LIN {X 0,Y 426.116,Z 779.168,A -85,B 0,C 180,E1 -10324.509,E2 -10324.509} C_VEL
LIN {X 0,Y 425.527,Z 793.819,A -85,B 0,C 180,E1 -10324.947,E2 -10324.947} C_VEL
LIN {X 0,Y 424.719,Z 807.739,A -85,B 0,C 180,E1 -10325.563,E2 -10325.563} C_VEL
LIN {X 0,Y 423.969,Z 820.23,A -85,B 0,C 180,E1 -10326.308,E2 -10326.308} C_VEL
LIN {X 0,Y 422.947,Z 832.999,A -85,B 0,C 180,E1 -10327.273,E2 -10327.273} C_VEL
LIN {X 0,Y 422.02,Z 844.698,A -85,B 0,C 180,E1 -10328.38,E2 -10328.38} C_VEL
LIN {X 0,Y 421.156,Z 854.395,A -85,B 0,C 180,E1 -10329.486,E2 -10329.486} C_VEL
LIN {X 0,Y 420.11,Z 865.116,A -85,B 0,C 180,E1 -10330.961,E2 -10330.961} C_VEL
LIN {X 0,Y 419.261,Z 873.928,A -85,B 0,C 180,E1 -10332.438,E2 -10332.438} C_VEL
LIN {X 0,Y 418.634,Z 881.226,A -85,B 0,C 180,E1 -10333.919,E2 -10333.919} C_VEL
LIN {X 0,Y 417.959,Z 888.478,A -85,B 0,C 180,E1 -10335.723,E2 -10335.723} C_VEL
LIN {X 0,Y 417.146,Z 891.035,A -85,B 0,C 180,E1 -10336.445,E2 -10336.445} C_VEL
LIN {X 0,Y 414.039,Z 894.793,A -85,B 0,C 180,E1 -10337.635,E2 -10337.635} C_VEL
LIN {X 0,Y 411.432,Z 897.379,A -85,B 0,C 180,E1 -10338.619,E2 -10338.619} C_VEL
LIN {X 0,Y 410.263,Z 899.081,A -85,B 0,C 180,E1 -10339.397,E2 -10339.397} C_VEL
LIN {X 0,Y 410.139,Z 899.54,A -85,B 0,C 180,E1 -10339.664,E2 -10339.664} C_VEL
LIN {X 0,Y 410.039,Z 901.862,A -85,B 0,C 180,E1 -10341.126,E2 -10341.126} C_VEL
LIN {X 0,Y 410.034,Z 903.737,A -85,B 0,C 180,E1 -10343.109,E2 -10343.109} C_VEL
LIN {X 0,Y 409.968,Z 904.281,A -85,B 0,C 180,E1 -10345.083,E2 -10345.083} C_VEL
LIN {X 0,Y 409.988,Z 903.511,A -85,B 0,C 180,E1 -10347.052,E2 -10347.052} C_VEL
LIN {X 0,Y 410.005,Z 901.424,A -85,B 0,C 180,E1 -10349.018,E2 -10349.018} C_VEL
LIN {X 0,Y 410.11,Z 897.97,A -85,B 0,C 180,E1 -10350.982,E2 -10350.982} C_VEL
LIN {X 0,Y 410.446,Z 893.043,A -85,B 0,C 180,E1 -10352.945,E2 -10352.945} C_VEL
LIN {X 0,Y 411.09,Z 886.486,A -85,B 0,C 180,E1 -10354.904,E2 -10354.904} C_VEL
LIN {X 0,Y 411.743,Z 879.197,A -85,B 0,C 180,E1 -10356.616,E2 -10356.616} C_VEL
LIN {X 0,Y 412.336,Z 870.804,A -85,B 0,C 180,E1 -10358.222,E2 -10358.222} C_VEL
LIN {X 0,Y 413.209,Z 861.976,A -85,B 0,C 180,E1 -10359.614,E2 -10359.614} C_VEL
LIN {X 0,Y 414.215,Z 851.288,A -85,B 0,C 180,E1 -10361.004,E2 -10361.004} C_VEL
LIN {X 0,Y 415.185,Z 839.942,A -85,B 0,C 180,E1 -10362.216,E2 -10362.216} C_VEL
LIN {X 0,Y 416.148,Z 827.376,A -85,B 0,C 180,E1 -10363.303,E2 -10363.303} C_VEL
LIN {X 0,Y 416.988,Z 815.158,A -85,B 0,C 180,E1 -10364.146,E2 -10364.146} C_VEL
LIN {X 0,Y 417.734,Z 801.639,A -85,B 0,C 180,E1 -10364.867,E2 -10364.867} C_VEL
LIN {X 0,Y 418.279,Z 787.615,A -85,B 0,C 180,E1 -10365.408,E2 -10365.408} C_VEL
LIN {X 0,Y 418.632,Z 772.8,A -85,B 0,C 180,E1 -10365.769,E2 -10365.769} C_VEL
LIN {X 0,Y 420.223,Z 667.238,A -85,B 0,C 180,E1 -10367.579,E2 -10367.579} C_VEL
LIN {X 0,Y 416.862,Z 653.116,A -85,B 0,C 180,E1 -10368.014,E2 -10368.014} C_VEL
LIN {X 0,Y 413.362,Z 643.418,A -85,B 0,C 180,E1 -10368.406,E2 -10368.406} C_VEL
LIN {X 0,Y 411.214,Z 633.392,A -85,B 0,C 180,E1 -10370.775,E2 -10370.775} C_VEL
LIN {X 0,Y 411.193,Z 633.392,A -85,B 0,C 180,E1 -10374.218,E2 -10374.218} C_VEL
LIN {X 0,Y 411.145,Z 633.397,A -85,B 0,C 180,E1 -10377.486,E2 -10377.486} C_VEL
LIN {X 0,Y 411.197,Z 633.388,A -85,B 0,C 180,E1 -10379.713,E2 -10379.713} C_VEL
LIN {X 0,Y 411.206,Z 633.39,A -85,B 0,C 180,E1 -10383.156,E2 -10383.156} C_VEL
LIN {X 0,Y 411.192,Z 633.39,A -85,B 0,C 180,E1 -10386.551,E2 -10386.551} C_VEL
LIN {X 0,Y 411.171,Z 633.379,A -85,B 0,C 180,E1 -10389.72,E2 -10389.72} C_VEL
LIN {X 0,Y 411.165,Z 633.393,A -85,B 0,C 180,E1 -10393.135,E2 -10393.135} C_VEL
LIN {X 0,Y 411.167,Z 633.39,A -85,B 0,C 180,E1 -10395.882,E2 -10395.882} C_VEL
LIN {X 0,Y 411.161,Z 633.392,A -85,B 0,C 180,E1 -10399.493,E2 -10399.493} C_VEL
LIN {X 0,Y 411.186,Z 633.373,A -85,B 0,C 180,E1 -10402.025,E2 -10402.025} C_VEL
LIN {X 0,Y 411.207,Z 633.387,A -85,B 0,C 180,E1 -10405.666,E2 -10405.666} C_VEL
LIN {X 0,Y 411.192,Z 633.385,A -85,B 0,C 180,E1 -10409.152,E2 -10409.152} C_VEL
LIN {X 0,Y 411.183,Z 633.39,A -85,B 0,C 180,E1 -10411.407,E2 -10411.407} C_VEL
LIN {X 0,Y 411.215,Z 633.383,A -85,B 0,C 180,E1 -10414.934,E2 -10414.934} C_VEL
LIN {X 0,Y 411.206,Z 633.386,A -85,B 0,C 180,E1 -10417.913,E2 -10417.913} C_VEL
LIN {X 0,Y 411.223,Z 633.383,A -85,B 0,C 180,E1 -10421.051,E2 -10421.051} C_VEL
LIN {X 0,Y 411.257,Z 633.377,A -85,B 0,C 180,E1 -10424.131,E2 -10424.131} C_VEL
LIN {X 0,Y 411.307,Z 633.374,A -85,B 0,C 180,E1 -10427.165,E2 -10427.165} C_VEL
LIN {X 0,Y 411.294,Z 633.368,A -85,B 0,C 180,E1 -10430.161,E2 -10430.161} C_VEL
LIN {X 0,Y 411.396,Z 633.362,A -85,B 0,C 180,E1 -10433.132,E2 -10433.132} C_VEL
LIN {X 0,Y 411.305,Z 633.372,A -85,B 0,C 180,E1 -10435.099,E2 -10435.099} C_VEL
LIN {X 0,Y 411.512,Z 633.351,A -85,B 0,C 180,E1 -10438.042,E2 -10438.042} C_VEL
LIN {X 0,Y 411.641,Z 633.33,A -85,B 0,C 180,E1 -10440,E2 -10440} C_VEL
LIN {X 0,Y 411.459,Z 633.353,A -85,B 0,C 180,E1 -10442.937,E2 -10442.937} C_VEL
LIN {X 0,Y 411.432,Z 633.354,A -85,B 0,C 180,E1 -10446.867,E2 -10446.867} C_VEL
LIN {X 0,Y 411.295,Z 633.377,A -85,B 0,C 180,E1 -10449.838,E2 -10449.838} C_VEL
LIN {X 0,Y 411.308,Z 633.372,A -85,B 0,C 180,E1 -10453.104,E2 -10453.104} C_VEL
LIN {X 0,Y 411.267,Z 633.376,A -85,B 0,C 180,E1 -10456.869,E2 -10456.869} C_VEL
LIN {X 0,Y 411.233,Z 633.381,A -85,B 0,C 180,E1 -10459.986,E2 -10459.986} C_VEL
LIN {X 0,Y 411.198,Z 633.382,A -85,B 0,C 180,E1 -10463.148,E2 -10463.148} C_VEL
LIN {X 0,Y 411.238,Z 633.382,A -85,B 0,C 180,E1 -10466.381,E2 -10466.381} C_VEL
LIN {X 0,Y 411.202,Z 633.386,A -85,B 0,C 180,E1 -10469.712,E2 -10469.712} C_VEL
LIN {X 0,Y 411.208,Z 633.384,A -85,B 0,C 180,E1 -10473.155,E2 -10473.155} C_VEL
LIN {X 0,Y 411.197,Z 633.389,A -85,B 0,C 180,E1 -10476.553,E2 -10476.553} C_VEL
LIN {X 0,Y 411.228,Z 633.381,A -85,B 0,C 180,E1 -10479.73,E2 -10479.73} C_VEL
LIN {X 0,Y 411.178,Z 633.389,A -85,B 0,C 180,E1 -10483.133,E2 -10483.133} C_VEL
LIN {X 0,Y 411.174,Z 633.389,A -85,B 0,C 180,E1 -10485.88,E2 -10485.88} C_VEL
LIN {X 0,Y 411.167,Z 633.394,A -85,B 0,C 180,E1 -10488.771,E2 -10488.771} C_VEL
LIN {X 0,Y 411.213,Z 633.386,A -85,B 0,C 180,E1 -10491.83,E2 -10491.83} C_VEL
LIN {X 0,Y 411.213,Z 633.39,A -85,B 0,C 180,E1 -10495.121,E2 -10495.121} C_VEL
LIN {X 0,Y 411.167,Z 633.39,A -85,B 0,C 180,E1 -10498.003,E2 -10498.003} C_VEL
LIN {X 0,Y 411.262,Z 633.533,A -85,B 0,C 180,E1 -10499.372,E2 -10499.372} C_VEL
LIN {X 0,Y 414.549,Z 647.989,A -85,B 0,C 180,E1 -10502.318,E2 -10502.318} C_VEL
LIN {X 0,Y 415.856,Z 654.509,A -85,B 0,C 180,E1 -10503.599,E2 -10503.599} C_VEL
LIN {X 0,Y 414.842,Z 669.698,A -85,B 0,C 180,E1 -10506.317,E2 -10506.317} C_VEL
LIN {X 0,Y 414.706,Z 671.836,A -85,B 0,C 180,E1 -10506.696,E2 -10506.696} C_VEL
LIN {X 0,Y 419.881,Z 702.214,A -85,B 0,C 180,E1 -10507.528,E2 -10507.528} C_VEL
LIN {X 0,Y 418.525,Z 800.905,A -85,B 0,C 180,E1 -10509.223,E2 -10509.223} C_VEL
LIN {X 0,Y 418.065,Z 815.953,A -85,B 0,C 180,E1 -10509.552,E2 -10509.552} C_VEL
LIN {X 0,Y 417.398,Z 830.189,A -85,B 0,C 180,E1 -10510.064,E2 -10510.064} C_VEL
LIN {X 0,Y 416.641,Z 843.346,A -85,B 0,C 180,E1 -10510.731,E2 -10510.731} C_VEL
LIN {X 0,Y 415.764,Z 855.462,A -85,B 0,C 180,E1 -10511.521,E2 -10511.521} C_VEL
LIN {X 0,Y 414.818,Z 867.42,A -85,B 0,C 180,E1 -10512.499,E2 -10512.499} C_VEL
LIN {X 0,Y 413.753,Z 879.543,A -85,B 0,C 180,E1 -10513.724,E2 -10513.724} C_VEL
LIN {X 0,Y 412.833,Z 889.574,A -85,B 0,C 180,E1 -10514.953,E2 -10514.953} C_VEL
LIN {X 0,Y 411.997,Z 899.202,A -85,B 0,C 180,E1 -10516.373,E2 -10516.373} C_VEL
LIN {X 0,Y 411.326,Z 907.866,A -85,B 0,C 180,E1 -10517.918,E2 -10517.918} C_VEL
LIN {X 0,Y 410.685,Z 915.798,A -85,B 0,C 180,E1 -10519.648,E2 -10519.648} C_VEL
LIN {X 0,Y 410.353,Z 921.358,A -85,B 0,C 180,E1 -10521.133,E2 -10521.133} C_VEL
LIN {X 0,Y 410.085,Z 927.19,A -85,B 0,C 180,E1 -10523.11,E2 -10523.11} C_VEL
LIN {X 0,Y 409.995,Z 931.435,A -85,B 0,C 180,E1 -10525.083,E2 -10525.083} C_VEL
LIN {X 0,Y 409.934,Z 934.224,A -85,B 0,C 180,E1 -10527.052,E2 -10527.052} C_VEL
LIN {X 0,Y 409.991,Z 935.101,A -85,B 0,C 180,E1 -10528.035,E2 -10528.035} C_VEL
LIN {X 0,Y 409.946,Z 935.837,A -85,B 0,C 180,E1 -10530,E2 -10530} C_VEL
LIN {X 0,Y 409.99,Z 935.235,A -85,B 0,C 180,E1 -10531.965,E2 -10531.965} C_VEL
LIN {X 0,Y 409.924,Z 933.276,A -85,B 0,C 180,E1 -10533.932,E2 -10533.932} C_VEL
LIN {X 0,Y 410.042,Z 929.917,A -85,B 0,C 180,E1 -10535.903,E2 -10535.903} C_VEL
LIN {X 0,Y 410.188,Z 925.062,A -85,B 0,C 180,E1 -10537.878,E2 -10537.878} C_VEL
LIN {X 0,Y 410.612,Z 918.581,A -85,B 0,C 180,E1 -10539.855,E2 -10539.855} C_VEL
LIN {X 0,Y 411.17,Z 911.384,A -85,B 0,C 180,E1 -10541.586,E2 -10541.586} C_VEL
LIN {X 0,Y 411.87,Z 903.781,A -85,B 0,C 180,E1 -10543.083,E2 -10543.083} C_VEL
LIN {X 0,Y 412.602,Z 894.853,A -85,B 0,C 180,E1 -10544.551,E2 -10544.551} C_VEL
LIN {X 0,Y 413.688,Z 883.963,A -85,B 0,C 180,E1 -10546.025,E2 -10546.025} C_VEL
LIN {X 0,Y 414.754,Z 872.932,A -85,B 0,C 180,E1 -10547.25,E2 -10547.25} C_VEL
LIN {X 0,Y 415.898,Z 860.846,A -85,B 0,C 180,E1 -10548.345,E2 -10548.345} C_VEL
LIN {X 0,Y 416.982,Z 847.686,A -85,B 0,C 180,E1 -10549.292,E2 -10549.292} C_VEL
LIN {X 0,Y 417.882,Z 834.246,A -85,B 0,C 180,E1 -10550.04,E2 -10550.04} C_VEL
LIN {X 0,Y 418.672,Z 820.158,A -85,B 0,C 180,E1 -10550.609,E2 -10550.609} C_VEL
LIN {X 0,Y 419.235,Z 805.296,A -85,B 0,C 180,E1 -10550.997,E2 -10550.997} C_VEL
LIN {X 0,Y 420.84,Z 702.534,A -85,B 0,C 180,E1 -10552.785,E2 -10552.785} C_VEL
LIN {X 0,Y 416.253,Z 677.29,A -85,B 0,C 180,E1 -10553.539,E2 -10553.539} C_VEL
LIN {X 0,Y 415.169,Z 671.541,A -85,B 0,C 180,E1 -10553.744,E2 -10553.744} C_VEL
LIN {X 0,Y 416.408,Z 657.156,A -85,B 0,C 180,E1 -10556.357,E2 -10556.357} C_VEL
LIN {X 0,Y 415.295,Z 650.459,A -85,B 0,C 180,E1 -10557.704,E2 -10557.704} C_VEL
LIN {X 0,Y 412.202,Z 637.376,A -85,B 0,C 180,E1 -10560.484,E2 -10560.484} C_VEL
LIN {X 0,Y 411.169,Z 633.391,A -85,B 0,C 180,E1 -10561.395,E2 -10561.395} C_VEL
LIN {X 0,Y 411.207,Z 633.383,A -85,B 0,C 180,E1 -10564.333,E2 -10564.333} C_VEL
LIN {X 0,Y 411.203,Z 633.386,A -85,B 0,C 180,E1 -10567.973,E2 -10567.973} C_VEL
LIN {X 0,Y 411.201,Z 633.385,A -85,B 0,C 180,E1 -10571.234,E2 -10571.234} C_VEL
LIN {X 0,Y 411.18,Z 633.385,A -85,B 0,C 180,E1 -10574.49,E2 -10574.49} C_VEL
LIN {X 0,Y 411.199,Z 633.38,A -85,B 0,C 180,E1 -10578.197,E2 -10578.197} C_VEL
LIN {X 0,Y 411.232,Z 633.383,A -85,B 0,C 180,E1 -10580.778,E2 -10580.778} C_VEL
LIN {X 0,Y 411.201,Z 633.385,A -85,B 0,C 180,E1 -10584.472,E2 -10584.472} C_VEL
LIN {X 0,Y 411.207,Z 633.382,A -85,B 0,C 180,E1 -10586.873,E2 -10586.873} C_VEL
LIN {X 0,Y 411.233,Z 633.379,A -85,B 0,C 180,E1 -10590.644,E2 -10590.644} C_VEL
LIN {X 0,Y 411.239,Z 633.381,A -85,B 0,C 180,E1 -10593.619,E2 -10593.619} C_VEL
LIN {X 0,Y 411.204,Z 633.382,A -85,B 0,C 180,E1 -10596.853,E2 -10596.853} C_VEL
LIN {X 0,Y 411.217,Z 633.388,A -85,B 0,C 180,E1 -10600.05,E2 -10600.05} C_VEL
LIN {X 0,Y 411.266,Z 633.377,A -85,B 0,C 180,E1 -10603.131,E2 -10603.131} C_VEL
LIN {X 0,Y 411.307,Z 633.37,A -85,B 0,C 180,E1 -10606.896,E2 -10606.896} C_VEL
LIN {X 0,Y 411.295,Z 633.373,A -85,B 0,C 180,E1 -10610.162,E2 -10610.162} C_VEL
LIN {X 0,Y 411.454,Z 633.354,A -85,B 0,C 180,E1 -10613.133,E2 -10613.133} C_VEL
LIN {X 0,Y 411.311,Z 633.367,A -85,B 0,C 180,E1 -10615.099,E2 -10615.099} C_VEL
LIN {X 0,Y 411.513,Z 633.35,A -85,B 0,C 180,E1 -10618.043,E2 -10618.043} C_VEL
LIN {X 0,Y 411.642,Z 633.332,A -85,B 0,C 180,E1 -10620,E2 -10620} C_VEL
LIN {X 0,Y 411.459,Z 633.355,A -85,B 0,C 180,E1 -10622.938,E2 -10622.938} C_VEL
LIN {X 0,Y 411.453,Z 633.357,A -85,B 0,C 180,E1 -10626.867,E2 -10626.867} C_VEL
LIN {X 0,Y 411.294,Z 633.372,A -85,B 0,C 180,E1 -10629.839,E2 -10629.839} C_VEL
LIN {X 0,Y 411.308,Z 633.373,A -85,B 0,C 180,E1 -10633.105,E2 -10633.105} C_VEL
LIN {X 0,Y 411.265,Z 633.383,A -85,B 0,C 180,E1 -10636.869,E2 -10636.869} C_VEL
LIN {X 0,Y 411.233,Z 633.377,A -85,B 0,C 180,E1 -10639.987,E2 -10639.987} C_VEL
LIN {X 0,Y 411.198,Z 633.384,A -85,B 0,C 180,E1 -10643.148,E2 -10643.148} C_VEL
LIN {X 0,Y 411.198,Z 633.389,A -85,B 0,C 180,E1 -10646.384,E2 -10646.384} C_VEL
LIN {X 0,Y 411.2,Z 633.374,A -85,B 0,C 180,E1 -10649.713,E2 -10649.713} C_VEL
LIN {X 0,Y 411.209,Z 633.386,A -85,B 0,C 180,E1 -10653.156,E2 -10653.156} C_VEL
LIN {X 0,Y 411.194,Z 633.389,A -85,B 0,C 180,E1 -10656.553,E2 -10656.553} C_VEL
LIN {X 0,Y 411.18,Z 633.384,A -85,B 0,C 180,E1 -10659.722,E2 -10659.722} C_VEL
LIN {X 0,Y 411.167,Z 633.397,A -85,B 0,C 180,E1 -10663.135,E2 -10663.135} C_VEL
LIN {X 0,Y 411.166,Z 633.389,A -85,B 0,C 180,E1 -10665.882,E2 -10665.882} C_VEL
LIN {X 0,Y 411.165,Z 633.397,A -85,B 0,C 180,E1 -10669.494,E2 -10669.494} C_VEL
LIN {X 0,Y 411.19,Z 633.391,A -85,B 0,C 180,E1 -10672.026,E2 -10672.026} C_VEL
LIN {X 0,Y 411.196,Z 633.39,A -85,B 0,C 180,E1 -10675.666,E2 -10675.666} C_VEL
LIN {X 0,Y 411.209,Z 633.511,A -85,B 0,C 180,E1 -10678.711,E2 -10678.711} C_VEL
LIN {X 0,Y 413.516,Z 643.651,A -85,B 0,C 180,E1 -10681.219,E2 -10681.219} C_VEL
LIN {X 0,Y 418.909,Z 657.328,A -85,B 0,C 180,E1 -10681.84,E2 -10681.84} C_VEL
LIN {X 0,Y 421.274,Z 668.298,A -85,B 0,C 180,E1 -10682.193,E2 -10682.193} C_VEL
LIN {X 0,Y 419.565,Z 779.554,A -85,B 0,C 180,E1 -10684.149,E2 -10684.149} C_VEL
LIN {X 0,Y 418.987,Z 793.733,A -85,B 0,C 180,E1 -10684.577,E2 -10684.577} C_VEL
LIN {X 0,Y 418.213,Z 806.917,A -85,B 0,C 180,E1 -10685.158,E2 -10685.158} C_VEL
LIN {X 0,Y 417.367,Z 819.977,A -85,B 0,C 180,E1 -10685.935,E2 -10685.935} C_VEL
LIN {X 0,Y 416.313,Z 832.576,A -85,B 0,C 180,E1 -10686.89,E2 -10686.89} C_VEL
LIN {X 0,Y 415.287,Z 844.394,A -85,B 0,C 180,E1 -10688.011,E2 -10688.011} C_VEL
LIN {X 0,Y 414.397,Z 854.189,A -85,B 0,C 180,E1 -10689.136,E2 -10689.136} C_VEL
LIN {X 0,Y 413.297,Z 864.988,A -85,B 0,C 180,E1 -10690.635,E2 -10690.635} C_VEL
LIN {X 0,Y 412.366,Z 873.867,A -85,B 0,C 180,E1 -10692.135,E2 -10692.135} C_VEL
LIN {X 0,Y 411.691,Z 881.223,A -85,B 0,C 180,E1 -10693.64,E2 -10693.64} C_VEL
LIN {X 0,Y 411.075,Z 887.322,A -85,B 0,C 180,E1 -10695.141,E2 -10695.141} C_VEL
LIN {X 0,Y 410.691,Z 892.354,A -85,B 0,C 180,E1 -10696.643,E2 -10696.643} C_VEL
LIN {X 0,Y 410.304,Z 897.512,A -85,B 0,C 180,E1 -10698.64,E2 -10698.64} C_VEL
LIN {X 0,Y 410.139,Z 899.54,A -85,B 0,C 180,E1 -10699.664,E2 -10699.664} C_VEL
LIN {X 0,Y 409.406,Z 900.948,A -85,B 0,C 180,E1 -10700.459,E2 -10700.459} C_VEL
LIN {X 0,Y 406.562,Z 902.765,A -85,B 0,C 180,E1 -10701.765,E2 -10701.765} C_VEL
LIN {X 0,Y 404.149,Z 903.807,A -85,B 0,C 180,E1 -10702.829,E2 -10702.829} C_VEL
LIN {X 0,Y 403.043,Z 904.3,A -85,B 0,C 180,E1 -10703.655,E2 -10703.655} C_VEL
LIN {X 0,Y 402.912,Z 904.415,A -85,B 0,C 180,E1 -10703.935,E2 -10703.935} C_VEL
LIN {X 0,Y 402.838,Z 904.364,A -85,B 0,C 180,E1 -10705.998,E2 -10705.998} C_VEL
LIN {X 0,Y 402.959,Z 902.973,A -85,B 0,C 180,E1 -10708.001,E2 -10708.001} C_VEL
LIN {X 0,Y 402.947,Z 900.255,A -85,B 0,C 180,E1 -10710,E2 -10710} C_VEL
LIN {X 0,Y 403.191,Z 897.316,A -85,B 0,C 180,E1 -10711.498,E2 -10711.498} C_VEL
LIN {X 0,Y 403.618,Z 892.036,A -85,B 0,C 180,E1 -10713.494,E2 -10713.494} C_VEL
LIN {X 0,Y 404.05,Z 886.977,A -85,B 0,C 180,E1 -10714.989,E2 -10714.989} C_VEL
LIN {X 0,Y 404.729,Z 879.746,A -85,B 0,C 180,E1 -10716.731,E2 -10716.731} C_VEL
LIN {X 0,Y 405.318,Z 871.709,A -85,B 0,C 180,E1 -10718.314,E2 -10718.314} C_VEL
LIN {X 0,Y 406.177,Z 863.265,A -85,B 0,C 180,E1 -10719.687,E2 -10719.687} C_VEL
LIN {X 0,Y 407.117,Z 854.045,A -85,B 0,C 180,E1 -10720.947,E2 -10720.947} C_VEL
LIN {X 0,Y 408.115,Z 843.248,A -85,B 0,C 180,E1 -10722.178,E2 -10722.178} C_VEL
LIN {X 0,Y 409.041,Z 831.435,A -85,B 0,C 180,E1 -10723.286,E2 -10723.286} C_VEL
LIN {X 0,Y 410.04,Z 818.329,A -85,B 0,C 180,E1 -10724.264,E2 -10724.264} C_VEL
LIN {X 0,Y 410.89,Z 804.421,A -85,B 0,C 180,E1 -10725.057,E2 -10725.057} C_VEL
LIN {X 0,Y 411.522,Z 790.504,A -85,B 0,C 180,E1 -10725.635,E2 -10725.635} C_VEL
LIN {X 0,Y 411.884,Z 775.94,A -85,B 0,C 180,E1 -10726.034,E2 -10726.034} C_VEL
LIN {X 0,Y 413.626,Z 668.286,A -85,B 0,C 180,E1 -10727.915,E2 -10727.915} C_VEL
LIN {X 0,Y 410.4,Z 655.06,A -85,B 0,C 180,E1 -10728.336,E2 -10728.336} C_VEL
LIN {X 0,Y 406.21,Z 643.728,A -85,B 0,C 180,E1 -10728.802,E2 -10728.802} C_VEL
LIN {X 0,Y 404.161,Z 634.27,A -85,B 0,C 180,E1 -10731.084,E2 -10731.084} C_VEL
LIN {X 0,Y 404.152,Z 634.268,A -85,B 0,C 180,E1 -10733.576,E2 -10733.576} C_VEL
LIN {X 0,Y 404.1,Z 634.275,A -85,B 0,C 180,E1 -10736.884,E2 -10736.884} C_VEL
LIN {X 0,Y 404.144,Z 634.269,A -85,B 0,C 180,E1 -10740.285,E2 -10740.285} C_VEL
LIN {X 0,Y 404.139,Z 634.267,A -85,B 0,C 180,E1 -10743.813,E2 -10743.813} C_VEL
LIN {X 0,Y 404.135,Z 634.271,A -85,B 0,C 180,E1 -10746.874,E2 -10746.874} C_VEL
LIN {X 0,Y 404.12,Z 634.256,A -85,B 0,C 180,E1 -10750.075,E2 -10750.075} C_VEL
LIN {X 0,Y 404.145,Z 634.268,A -85,B 0,C 180,E1 -10753.082,E2 -10753.082} C_VEL
LIN {X 0,Y 404.123,Z 634.267,A -85,B 0,C 180,E1 -10755.922,E2 -10755.922} C_VEL
LIN {X 0,Y 404.104,Z 634.271,A -85,B 0,C 180,E1 -10758.632,E2 -10758.632} C_VEL
LIN {X 0,Y 404.141,Z 634.254,A -85,B 0,C 180,E1 -10761.495,E2 -10761.495} C_VEL
LIN {X 0,Y 404.182,Z 634.255,A -85,B 0,C 180,E1 -10764.983,E2 -10764.983} C_VEL
LIN {X 0,Y 404.142,Z 634.263,A -85,B 0,C 180,E1 -10768.442,E2 -10768.442} C_VEL
LIN {X 0,Y 404.156,Z 634.259,A -85,B 0,C 180,E1 -10770.862,E2 -10770.862} C_VEL
LIN {X 0,Y 404.141,Z 634.262,A -85,B 0,C 180,E1 -10774.23,E2 -10774.23} C_VEL
LIN {X 0,Y 404.169,Z 634.262,A -85,B 0,C 180,E1 -10777.508,E2 -10777.508} C_VEL
LIN {X 0,Y 404.166,Z 634.26,A -85,B 0,C 180,E1 -10780.707,E2 -10780.707} C_VEL
LIN {X 0,Y 404.224,Z 634.255,A -85,B 0,C 180,E1 -10783.848,E2 -10783.848} C_VEL
LIN {X 0,Y 404.286,Z 634.247,A -85,B 0,C 180,E1 -10786.939,E2 -10786.939} C_VEL
LIN {X 0,Y 404.259,Z 634.244,A -85,B 0,C 180,E1 -10789.988,E2 -10789.988} C_VEL
LIN {X 0,Y 404.346,Z 634.24,A -85,B 0,C 180,E1 -10793.011,E2 -10793.011} C_VEL
LIN {X 0,Y 404.275,Z 634.247,A -85,B 0,C 180,E1 -10795.013,E2 -10795.013} C_VEL
LIN {X 0,Y 404.481,Z 634.227,A -85,B 0,C 180,E1 -10798.008,E2 -10798.008} C_VEL
LIN {X 0,Y 404.61,Z 634.206,A -85,B 0,C 180,E1 -10800,E2 -10800} C_VEL
LIN {X 0,Y 404.417,Z 634.23,A -85,B 0,C 180,E1 -10802.988,E2 -10802.988} C_VEL
LIN {X 0,Y 404.382,Z 634.233,A -85,B 0,C 180,E1 -10806.987,E2 -10806.987} C_VEL
LIN {X 0,Y 404.26,Z 634.251,A -85,B 0,C 180,E1 -10810.011,E2 -10810.011} C_VEL
LIN {X 0,Y 404.269,Z 634.249,A -85,B 0,C 180,E1 -10813.211,E2 -10813.211} C_VEL
LIN {X 0,Y 404.221,Z 634.253,A -85,B 0,C 180,E1 -10817.008,E2 -10817.008} C_VEL
LIN {X 0,Y 404.166,Z 634.264,A -85,B 0,C 180,E1 -10820.351,E2 -10820.351} C_VEL
LIN {X 0,Y 404.165,Z 634.259,A -85,B 0,C 180,E1 -10823.575,E2 -10823.575} C_VEL
LIN {X 0,Y 404.185,Z 634.261,A -85,B 0,C 180,E1 -10825.766,E2 -10825.766} C_VEL
LIN {X 0,Y 404.197,Z 634.258,A -85,B 0,C 180,E1 -10827.999,E2 -10827.999} C_VEL
LIN {X 0,Y 404.141,Z 634.264,A -85,B 0,C 180,E1 -10831.558,E2 -10831.558} C_VEL
LIN {X 0,Y 404.187,Z 634.261,A -85,B 0,C 180,E1 -10835.016,E2 -10835.016} C_VEL
LIN {X 0,Y 404.164,Z 634.264,A -85,B 0,C 180,E1 -10838.756,E2 -10838.756} C_VEL
LIN {X 0,Y 404.151,Z 634.263,A -85,B 0,C 180,E1 -10841.604,E2 -10841.604} C_VEL
LIN {X 0,Y 404.148,Z 634.268,A -85,B 0,C 180,E1 -10844.522,E2 -10844.522} C_VEL
LIN {X 0,Y 404.141,Z 634.264,A -85,B 0,C 180,E1 -10847.296,E2 -10847.296} C_VEL
LIN {X 0,Y 404.17,Z 634.264,A -85,B 0,C 180,E1 -10849.955,E2 -10849.955} C_VEL
LIN {X 0,Y 404.141,Z 634.27,A -85,B 0,C 180,E1 -10853.124,E2 -10853.124} C_VEL
LIN {X 0,Y 404.146,Z 634.268,A -85,B 0,C 180,E1 -10856.188,E2 -10856.188} C_VEL
LIN {X 0,Y 404.172,Z 634.354,A -85,B 0,C 180,E1 -10859.029,E2 -10859.029} C_VEL
LIN {X 0,Y 407.346,Z 647.988,A -85,B 0,C 180,E1 -10861.876,E2 -10861.876} C_VEL
LIN {X 0,Y 408.945,Z 655.881,A -85,B 0,C 180,E1 -10863.459,E2 -10863.459} C_VEL
LIN {X 0,Y 408.024,Z 669.316,A -85,B 0,C 180,E1 -10865.909,E2 -10865.909} C_VEL
LIN {X 0,Y 407.839,Z 671.559,A -85,B 0,C 180,E1 -10866.313,E2 -10866.313} C_VEL
LIN {X 0,Y 413.265,Z 703.387,A -85,B 0,C 180,E1 -10867.204,E2 -10867.204} C_VEL
LIN {X 0,Y 411.827,Z 800.85,A -85,B 0,C 180,E1 -10868.901,E2 -10868.901} C_VEL
LIN {X 0,Y 411.354,Z 815.82,A -85,B 0,C 180,E1 -10869.236,E2 -10869.236} C_VEL
LIN {X 0,Y 410.714,Z 829.32,A -85,B 0,C 180,E1 -10869.726,E2 -10869.726} C_VEL
LIN {X 0,Y 409.861,Z 843.302,A -85,B 0,C 180,E1 -10870.442,E2 -10870.442} C_VEL
LIN {X 0,Y 408.859,Z 856.439,A -85,B 0,C 180,E1 -10871.328,E2 -10871.328} C_VEL
LIN {X 0,Y 407.75,Z 869.471,A -85,B 0,C 180,E1 -10872.444,E2 -10872.444} C_VEL
LIN {X 0,Y 406.78,Z 880.119,A -85,B 0,C 180,E1 -10873.566,E2 -10873.566} C_VEL
LIN {X 0,Y 405.73,Z 890.909,A -85,B 0,C 180,E1 -10874.94,E2 -10874.94} C_VEL
LIN {X 0,Y 404.825,Z 900.701,A -85,B 0,C 180,E1 -10876.456,E2 -10876.456} C_VEL
LIN {X 0,Y 404.221,Z 908.709,A -85,B 0,C 180,E1 -10877.957,E2 -10877.957} C_VEL
LIN {X 0,Y 403.571,Z 916.44,A -85,B 0,C 180,E1 -10879.718,E2 -10879.718} C_VEL
LIN {X 0,Y 403.191,Z 922.635,A -85,B 0,C 180,E1 -10881.479,E2 -10881.479} C_VEL
LIN {X 0,Y 403.005,Z 926.854,A -85,B 0,C 180,E1 -10882.988,E2 -10882.988} C_VEL
LIN {X 0,Y 402.985,Z 929.177,A -85,B 0,C 180,E1 -10883.994,E2 -10883.994} C_VEL
LIN {X 0,Y 402.844,Z 932.695,A -85,B 0,C 180,E1 -10885.998,E2 -10885.998} C_VEL
LIN {X 0,Y 402.902,Z 934.809,A -85,B 0,C 180,E1 -10888.001,E2 -10888.001} C_VEL
LIN {X 0,Y 402.869,Z 935.56,A -85,B 0,C 180,E1 -10890,E2 -10890} C_VEL
LIN {X 0,Y 402.9,Z 934.975,A -85,B 0,C 180,E1 -10891.999,E2 -10891.999} C_VEL
LIN {X 0,Y 402.844,Z 933.036,A -85,B 0,C 180,E1 -10894.001,E2 -10894.001} C_VEL
LIN {X 0,Y 402.965,Z 929.695,A -85,B 0,C 180,E1 -10896.007,E2 -10896.007} C_VEL
LIN {X 0,Y 403.134,Z 924.859,A -85,B 0,C 180,E1 -10898.017,E2 -10898.017} C_VEL
LIN {X 0,Y 403.546,Z 918.397,A -85,B 0,C 180,E1 -10900.029,E2 -10900.029} C_VEL
LIN {X 0,Y 404.179,Z 911.224,A -85,B 0,C 180,E1 -10901.789,E2 -10901.789} C_VEL
LIN {X 0,Y 404.992,Z 902.792,A -85,B 0,C 180,E1 -10903.47,E2 -10903.47} C_VEL
LIN {X 0,Y 405.873,Z 893.119,A -85,B 0,C 180,E1 -10905.054,E2 -10905.054} C_VEL
LIN {X 0,Y 406.944,Z 882.918,A -85,B 0,C 180,E1 -10906.427,E2 -10906.427} C_VEL
LIN {X 0,Y 408.113,Z 871.716,A -85,B 0,C 180,E1 -10907.669,E2 -10907.669} C_VEL
LIN {X 0,Y 409.301,Z 859.358,A -85,B 0,C 180,E1 -10908.781,E2 -10908.781} C_VEL
LIN {X 0,Y 410.359,Z 846.757,A -85,B 0,C 180,E1 -10909.688,E2 -10909.688} C_VEL
LIN {X 0,Y 411.31,Z 833.251,A -85,B 0,C 180,E1 -10910.439,E2 -10910.439} C_VEL
LIN {X 0,Y 412.167,Z 818.873,A -85,B 0,C 180,E1 -10911.015,E2 -10911.015} C_VEL
LIN {X 0,Y 412.71,Z 804.862,A -85,B 0,C 180,E1 -10911.378,E2 -10911.378} C_VEL
LIN {X 0,Y 414.39,Z 703.771,A -85,B 0,C 180,E1 -10913.162,E2 -10913.162} C_VEL
LIN {X 0,Y 410.065,Z 679.599,A -85,B 0,C 180,E1 -10913.897,E2 -10913.897} C_VEL
LIN {X 0,Y 408.445,Z 671.319,A -85,B 0,C 180,E1 -10914.182,E2 -10914.182} C_VEL
LIN {X 0,Y 409.566,Z 658.811,A -85,B 0,C 180,E1 -10916.497,E2 -10916.497} C_VEL
LIN {X 0,Y 408.332,Z 651.68,A -85,B 0,C 180,E1 -10917.963,E2 -10917.963} C_VEL
LIN {X 0,Y 405.649,Z 640.193,A -85,B 0,C 180,E1 -10920.449,E2 -10920.449} C_VEL
LIN {X 0,Y 404.121,Z 634.267,A -85,B 0,C 180,E1 -10921.824,E2 -10921.824} C_VEL
LIN {X 0,Y 404.183,Z 634.255,A -85,B 0,C 180,E1 -10925.19,E2 -10925.19} C_VEL
LIN {X 0,Y 404.162,Z 634.263,A -85,B 0,C 180,E1 -10928.756,E2 -10928.756} C_VEL
LIN {X 0,Y 404.151,Z 634.268,A -85,B 0,C 180,E1 -10931.604,E2 -10931.604} C_VEL
LIN {X 0,Y 404.149,Z 634.261,A -85,B 0,C 180,E1 -10934.523,E2 -10934.523} C_VEL
LIN {X 0,Y 404.171,Z 634.257,A -85,B 0,C 180,E1 -10937.3,E2 -10937.3} C_VEL
LIN {X 0,Y 404.169,Z 634.266,A -85,B 0,C 180,E1 -10939.955,E2 -10939.955} C_VEL
LIN {X 0,Y 404.141,Z 634.253,A -85,B 0,C 180,E1 -10943.124,E2 -10943.124} C_VEL
LIN {X 0,Y 404.146,Z 634.264,A -85,B 0,C 180,E1 -10946.188,E2 -10946.188} C_VEL
LIN {X 0,Y 404.146,Z 634.253,A -85,B 0,C 180,E1 -10949.715,E2 -10949.715} C_VEL
LIN {X 0,Y 404.196,Z 634.257,A -85,B 0,C 180,E1 -10953.123,E2 -10953.123} C_VEL
LIN {X 0,Y 404.178,Z 634.26,A -85,B 0,C 180,E1 -10955.335,E2 -10955.335} C_VEL
LIN {X 0,Y 404.14,Z 634.265,A -85,B 0,C 180,E1 -10958.581,E2 -10958.581} C_VEL
LIN {X 0,Y 404.212,Z 634.255,A -85,B 0,C 180,E1 -10961.762,E2 -10961.762} C_VEL
LIN {X 0,Y 404.213,Z 634.255,A -85,B 0,C 180,E1 -10964.883,E2 -10964.883} C_VEL
LIN {X 0,Y 404.258,Z 634.253,A -85,B 0,C 180,E1 -10967.959,E2 -10967.959} C_VEL
LIN {X 0,Y 404.406,Z 634.233,A -85,B 0,C 180,E1 -10972.129,E2 -10972.129} C_VEL
LIN {X 0,Y 404.422,Z 634.235,A -85,B 0,C 180,E1 -10974.015,E2 -10974.015} C_VEL
LIN {X 0,Y 404.481,Z 634.226,A -85,B 0,C 180,E1 -10978.009,E2 -10978.009} C_VEL
LIN {X 0,Y 404.611,Z 634.207,A -85,B 0,C 180,E1 -10980,E2 -10980} C_VEL
LIN {X 0,Y 404.417,Z 634.232,A -85,B 0,C 180,E1 -10982.989,E2 -10982.989} C_VEL
LIN {X 0,Y 404.394,Z 634.231,A -85,B 0,C 180,E1 -10986.584,E2 -10986.584} C_VEL
LIN {X 0,Y 404.292,Z 634.245,A -85,B 0,C 180,E1 -10989.001,E2 -10989.001} C_VEL
LIN {X 0,Y 404.258,Z 634.25,A -85,B 0,C 180,E1 -10992.042,E2 -10992.042} C_VEL
LIN {X 0,Y 404.209,Z 634.254,A -85,B 0,C 180,E1 -10995.118,E2 -10995.118} C_VEL
LIN {X 0,Y 404.211,Z 634.259,A -85,B 0,C 180,E1 -10998.238,E2 -10998.238} C_VEL
LIN {X 0,Y 404.14,Z 634.266,A -85,B 0,C 180,E1 -11001.42,E2 -11001.42} C_VEL
LIN {X 0,Y 404.171,Z 634.263,A -85,B 0,C 180,E1 -11004.666,E2 -11004.666} C_VEL
LIN {X 0,Y 404.133,Z 634.257,A -85,B 0,C 180,E1 -11008.005,E2 -11008.005} C_VEL
LIN {X 0,Y 404.146,Z 634.253,A -85,B 0,C 180,E1 -11010.286,E2 -11010.286} C_VEL
LIN {X 0,Y 404.146,Z 634.261,A -85,B 0,C 180,E1 -11013.813,E2 -11013.813} C_VEL
LIN {X 0,Y 404.137,Z 634.268,A -85,B 0,C 180,E1 -11016.875,E2 -11016.875} C_VEL
LIN {X 0,Y 404.119,Z 634.263,A -85,B 0,C 180,E1 -11020.075,E2 -11020.075} C_VEL
LIN {X 0,Y 404.146,Z 634.271,A -85,B 0,C 180,E1 -11023.083,E2 -11023.083} C_VEL
LIN {X 0,Y 404.123,Z 634.267,A -85,B 0,C 180,E1 -11025.923,E2 -11025.923} C_VEL
LIN {X 0,Y 404.106,Z 634.274,A -85,B 0,C 180,E1 -11028.633,E2 -11028.633} C_VEL
LIN {X 0,Y 404.145,Z 634.271,A -85,B 0,C 180,E1 -11031.495,E2 -11031.495} C_VEL
LIN {X 0,Y 404.177,Z 634.262,A -85,B 0,C 180,E1 -11034.983,E2 -11034.983} C_VEL
LIN {X 0,Y 404.134,Z 634.392,A -85,B 0,C 180,E1 -11038.322,E2 -11038.322} C_VEL
LIN {X 0,Y 406.45,Z 644.112,A -85,B 0,C 180,E1 -11040.758,E2 -11040.758} C_VEL
LIN {X 0,Y 412.799,Z 659.86,A -85,B 0,C 180,E1 -11041.49,E2 -11041.49} C_VEL
LIN {X 0,Y 414.748,Z 668.607,A -85,B 0,C 180,E1 -11041.783,E2 -11041.783} C_VEL
LIN {X 0,Y 413.042,Z 779.979,A -85,B 0,C 180,E1 -11043.777,E2 -11043.777} C_VEL
LIN {X 0,Y 412.421,Z 794.09,A -85,B 0,C 180,E1 -11044.21,E2 -11044.21} C_VEL
LIN {X 0,Y 411.593,Z 807.659,A -85,B 0,C 180,E1 -11044.822,E2 -11044.822} C_VEL
LIN {X 0,Y 410.668,Z 821.106,A -85,B 0,C 180,E1 -11045.645,E2 -11045.645} C_VEL
LIN {X 0,Y 409.566,Z 833.604,A -85,B 0,C 180,E1 -11046.621,E2 -11046.621} C_VEL
LIN {X 0,Y 408.483,Z 845.285,A -85,B 0,C 180,E1 -11047.758,E2 -11047.758} C_VEL
LIN {X 0,Y 407.454,Z 855.957,A -85,B 0,C 180,E1 -11049.028,E2 -11049.028} C_VEL
LIN {X 0,Y 406.325,Z 866.505,A -85,B 0,C 180,E1 -11050.552,E2 -11050.552} C_VEL
LIN {X 0,Y 405.368,Z 875.179,A -85,B 0,C 180,E1 -11052.078,E2 -11052.078} C_VEL
LIN {X 0,Y 404.558,Z 883.436,A -85,B 0,C 180,E1 -11053.862,E2 -11053.862} C_VEL
LIN {X 0,Y 403.933,Z 889.186,A -85,B 0,C 180,E1 -11055.387,E2 -11055.387} C_VEL
LIN {X 0,Y 403.442,Z 894.95,A -85,B 0,C 180,E1 -11057.3,E2 -11057.3} C_VEL
LIN {X 0,Y 403.185,Z 898.717,A -85,B 0,C 180,E1 -11058.946,E2 -11058.946} C_VEL
LIN {X 0,Y 402.95,Z 902.051,A -85,B 0,C 180,E1 -11060.969,E2 -11060.969} C_VEL
LIN {X 0,Y 402.95,Z 903.977,A -85,B 0,C 180,E1 -11062.987,E2 -11062.987} C_VEL
LIN {X 0,Y 402.912,Z 904.415,A -85,B 0,C 180,E1 -11063.935,E2 -11063.935} C_VEL
LIN {X 0,Y 402.147,Z 904.626,A -85,B 0,C 180,E1 -11064.769,E2 -11064.769} C_VEL
LIN {X 0,Y 399.307,Z 904.502,A -85,B 0,C 180,E1 -11066.126,E2 -11066.126} C_VEL
LIN {X 0,Y 396.963,Z 903.929,A -85,B 0,C 180,E1 -11067.219,E2 -11067.219} C_VEL
LIN {X 0,Y 395.951,Z 903.208,A -85,B 0,C 180,E1 -11068.058,E2 -11068.058} C_VEL
LIN {X 0,Y 395.861,Z 902.881,A -85,B 0,C 180,E1 -11068.341,E2 -11068.341} C_VEL
LIN {X 0,Y 395.869,Z 900.635,A -85,B 0,C 180,E1 -11070,E2 -11070} C_VEL
LIN {X 0,Y 396.087,Z 896.544,A -85,B 0,C 180,E1 -11072.034,E2 -11072.034} C_VEL
LIN {X 0,Y 396.543,Z 892.5,A -85,B 0,C 180,E1 -11073.557,E2 -11073.557} C_VEL
LIN {X 0,Y 397.013,Z 887.464,A -85,B 0,C 180,E1 -11075.078,E2 -11075.078} C_VEL
LIN {X 0,Y 397.716,Z 880.282,A -85,B 0,C 180,E1 -11076.851,E2 -11076.851} C_VEL
LIN {X 0,Y 398.308,Z 872.493,A -85,B 0,C 180,E1 -11078.425,E2 -11078.425} C_VEL
LIN {X 0,Y 399.233,Z 863.919,A -85,B 0,C 180,E1 -11079.858,E2 -11079.858} C_VEL
LIN {X 0,Y 400.38,Z 852.836,A -85,B 0,C 180,E1 -11081.389,E2 -11081.389} C_VEL
LIN {X 0,Y 401.424,Z 841.703,A -85,B 0,C 180,E1 -11082.641,E2 -11082.641} C_VEL
LIN {X 0,Y 402.476,Z 829.404,A -85,B 0,C 180,E1 -11083.764,E2 -11083.764} C_VEL
LIN {X 0,Y 403.367,Z 817.564,A -85,B 0,C 180,E1 -11084.634,E2 -11084.634} C_VEL
LIN {X 0,Y 404.196,Z 804.61,A -85,B 0,C 180,E1 -11085.377,E2 -11085.377} C_VEL
LIN {X 0,Y 404.839,Z 790.661,A -85,B 0,C 180,E1 -11085.965,E2 -11085.965} C_VEL
LIN {X 0,Y 405.225,Z 777.491,A -85,B 0,C 180,E1 -11086.337,E2 -11086.337} C_VEL
LIN {X 0,Y 406.934,Z 669.229,A -85,B 0,C 180,E1 -11088.268,E2 -11088.268} C_VEL
LIN {X 0,Y 404.126,Z 657.468,A -85,B 0,C 180,E1 -11088.649,E2 -11088.649} C_VEL
LIN {X 0,Y 399.046,Z 643.947,A -85,B 0,C 180,E1 -11089.234,E2 -11089.234} C_VEL
LIN {X 0,Y 397.136,Z 635.144,A -85,B 0,C 180,E1 -11091.407,E2 -11091.407} C_VEL
LIN {X 0,Y 397.105,Z 635.148,A -85,B 0,C 180,E1 -11095.135,E2 -11095.135} C_VEL
LIN {X 0,Y 397.064,Z 635.15,A -85,B 0,C 180,E1 -11098.548,E2 -11098.548} C_VEL
LIN {X 0,Y 397.078,Z 635.147,A -85,B 0,C 180,E1 -11101.835,E2 -11101.835} C_VEL
LIN {X 0,Y 397.118,Z 635.144,A -85,B 0,C 180,E1 -11104.494,E2 -11104.494} C_VEL
LIN {X 0,Y 397.093,Z 635.145,A -85,B 0,C 180,E1 -11108.276,E2 -11108.276} C_VEL
LIN {X 0,Y 397.054,Z 635.148,A -85,B 0,C 180,E1 -11111.976,E2 -11111.976} C_VEL
LIN {X 0,Y 397.089,Z 635.149,A -85,B 0,C 180,E1 -11115.069,E2 -11115.069} C_VEL
LIN {X 0,Y 397.054,Z 635.147,A -85,B 0,C 180,E1 -11118.023,E2 -11118.023} C_VEL
LIN {X 0,Y 397.093,Z 635.129,A -85,B 0,C 180,E1 -11121.723,E2 -11121.723} C_VEL
LIN {X 0,Y 397.125,Z 635.142,A -85,B 0,C 180,E1 -11125.506,E2 -11125.506} C_VEL
LIN {X 0,Y 397.081,Z 635.143,A -85,B 0,C 180,E1 -11129.117,E2 -11129.117} C_VEL
LIN {X 0,Y 397.085,Z 635.144,A -85,B 0,C 180,E1 -11132.246,E2 -11132.246} C_VEL
LIN {X 0,Y 397.114,Z 635.133,A -85,B 0,C 180,E1 -11135.98,E2 -11135.98} C_VEL
LIN {X 0,Y 397.142,Z 635.139,A -85,B 0,C 180,E1 -11139.704,E2 -11139.704} C_VEL
LIN {X 0,Y 397.185,Z 635.119,A -85,B 0,C 180,E1 -11142.845,E2 -11142.845} C_VEL
LIN {X 0,Y 397.232,Z 635.125,A -85,B 0,C 180,E1 -11146.702,E2 -11146.702} C_VEL
LIN {X 0,Y 397.219,Z 635.12,A -85,B 0,C 180,E1 -11149.809,E2 -11149.809} C_VEL
LIN {X 0,Y 397.298,Z 635.117,A -85,B 0,C 180,E1 -11152.887,E2 -11152.887} C_VEL
LIN {X 0,Y 397.245,Z 635.122,A -85,B 0,C 180,E1 -11154.925,E2 -11154.925} C_VEL
LIN {X 0,Y 397.45,Z 635.103,A -85,B 0,C 180,E1 -11157.973,E2 -11157.973} C_VEL
LIN {X 0,Y 397.58,Z 635.081,A -85,B 0,C 180,E1 -11160,E2 -11160} C_VEL
LIN {X 0,Y 397.377,Z 635.108,A -85,B 0,C 180,E1 -11163.041,E2 -11163.041} C_VEL
LIN {X 0,Y 397.335,Z 635.111,A -85,B 0,C 180,E1 -11167.112,E2 -11167.112} C_VEL
LIN {X 0,Y 397.22,Z 635.126,A -85,B 0,C 180,E1 -11170.191,E2 -11170.191} C_VEL
LIN {X 0,Y 397.229,Z 635.126,A -85,B 0,C 180,E1 -11173.321,E2 -11173.321} C_VEL
LIN {X 0,Y 397.174,Z 635.134,A -85,B 0,C 180,E1 -11176.446,E2 -11176.446} C_VEL
LIN {X 0,Y 397.15,Z 635.134,A -85,B 0,C 180,E1 -11179.647,E2 -11179.647} C_VEL
LIN {X 0,Y 397.114,Z 635.136,A -85,B 0,C 180,E1 -11183.032,E2 -11183.032} C_VEL
LIN {X 0,Y 397.136,Z 635.141,A -85,B 0,C 180,E1 -11186.258,E2 -11186.258} C_VEL
LIN {X 0,Y 397.124,Z 635.143,A -85,B 0,C 180,E1 -11188.543,E2 -11188.543} C_VEL
LIN {X 0,Y 397.08,Z 635.147,A -85,B 0,C 180,E1 -11192.071,E2 -11192.071} C_VEL
LIN {X 0,Y 397.121,Z 635.14,A -85,B 0,C 180,E1 -11195.503,E2 -11195.503} C_VEL
LIN {X 0,Y 397.138,Z 635.138,A -85,B 0,C 180,E1 -11198.862,E2 -11198.862} C_VEL
LIN {X 0,Y 397.115,Z 635.143,A -85,B 0,C 180,E1 -11202.261,E2 -11202.261} C_VEL
LIN {X 0,Y 397.091,Z 635.144,A -85,B 0,C 180,E1 -11205.068,E2 -11205.068} C_VEL
LIN {X 0,Y 397.07,Z 635.146,A -85,B 0,C 180,E1 -11208.02,E2 -11208.02} C_VEL
LIN {X 0,Y 397.135,Z 635.142,A -85,B 0,C 180,E1 -11211.138,E2 -11211.138} C_VEL
LIN {X 0,Y 397.121,Z 635.145,A -85,B 0,C 180,E1 -11214.496,E2 -11214.496} C_VEL
LIN {X 0,Y 397.079,Z 635.144,A -85,B 0,C 180,E1 -11217.928,E2 -11217.928} C_VEL
LIN {X 0,Y 397.109,Z 635.171,A -85,B 0,C 180,E1 -11218.676,E2 -11218.676} C_VEL
LIN {X 0,Y 400.44,Z 649.423,A -85,B 0,C 180,E1 -11221.714,E2 -11221.714} C_VEL
LIN {X 0,Y 402.012,Z 657.181,A -85,B 0,C 180,E1 -11223.301,E2 -11223.301} C_VEL
LIN {X 0,Y 401.698,Z 662.731,A -85,B 0,C 180,E1 -11224.34,E2 -11224.34} C_VEL
LIN {X 0,Y 401.009,Z 671.286,A -85,B 0,C 180,E1 -11225.919,E2 -11225.919} C_VEL
LIN {X 0,Y 406.646,Z 705.044,A -85,B 0,C 180,E1 -11226.878,E2 -11226.878} C_VEL
LIN {X 0,Y 404.947,Z 808.633,A -85,B 0,C 180,E1 -11228.725,E2 -11228.725} C_VEL
LIN {X 0,Y 404.36,Z 823.004,A -85,B 0,C 180,E1 -11229.16,E2 -11229.16} C_VEL
LIN {X 0,Y 403.54,Z 836.47,A -85,B 0,C 180,E1 -11229.762,E2 -11229.762} C_VEL
LIN {X 0,Y 402.648,Z 849.2,A -85,B 0,C 180,E1 -11230.524,E2 -11230.524} C_VEL
LIN {X 0,Y 401.574,Z 862.005,A -85,B 0,C 180,E1 -11231.506,E2 -11231.506} C_VEL
LIN {X 0,Y 400.432,Z 873.907,A -85,B 0,C 180,E1 -11232.64,E2 -11232.64} C_VEL
LIN {X 0,Y 399.374,Z 884.79,A -85,B 0,C 180,E1 -11233.909,E2 -11233.909} C_VEL
LIN {X 0,Y 398.27,Z 895.55,A -85,B 0,C 180,E1 -11235.436,E2 -11235.436} C_VEL
LIN {X 0,Y 397.605,Z 904.442,A -85,B 0,C 180,E1 -11236.975,E2 -11236.975} C_VEL
LIN {X 0,Y 396.826,Z 912.953,A -85,B 0,C 180,E1 -11238.766,E2 -11238.766} C_VEL
LIN {X 0,Y 396.344,Z 918.888,A -85,B 0,C 180,E1 -11240.302,E2 -11240.302} C_VEL
LIN {X 0,Y 396.001,Z 925.23,A -85,B 0,C 180,E1 -11242.351,E2 -11242.351} C_VEL
LIN {X 0,Y 395.908,Z 928.848,A -85,B 0,C 180,E1 -11243.886,E2 -11243.886} C_VEL
LIN {X 0,Y 395.766,Z 932.385,A -85,B 0,C 180,E1 -11245.927,E2 -11245.927} C_VEL
LIN {X 0,Y 395.815,Z 934.515,A -85,B 0,C 180,E1 -11247.965,E2 -11247.965} C_VEL
LIN {X 0,Y 395.795,Z 935.284,A -85,B 0,C 180,E1 -11250,E2 -11250} C_VEL
LIN {X 0,Y 395.797,Z 934.714,A -85,B 0,C 180,E1 -11252.035,E2 -11252.035} C_VEL
LIN {X 0,Y 395.766,Z 932.796,A -85,B 0,C 180,E1 -11254.073,E2 -11254.073} C_VEL
LIN {X 0,Y 395.908,Z 929.477,A -85,B 0,C 180,E1 -11256.114,E2 -11256.114} C_VEL
LIN {X 0,Y 396.07,Z 924.659,A -85,B 0,C 180,E1 -11258.161,E2 -11258.161} C_VEL
LIN {X 0,Y 396.383,Z 920.025,A -85,B 0,C 180,E1 -11259.697,E2 -11259.697} C_VEL
LIN {X 0,Y 396.986,Z 913.307,A -85,B 0,C 180,E1 -11261.488,E2 -11261.488} C_VEL
LIN {X 0,Y 397.815,Z 904.963,A -85,B 0,C 180,E1 -11263.277,E2 -11263.277} C_VEL
LIN {X 0,Y 398.608,Z 896.286,A -85,B 0,C 180,E1 -11264.812,E2 -11264.812} C_VEL
LIN {X 0,Y 399.779,Z 885.794,A -85,B 0,C 180,E1 -11266.336,E2 -11266.336} C_VEL
LIN {X 0,Y 400.954,Z 875.249,A -85,B 0,C 180,E1 -11267.599,E2 -11267.599} C_VEL
LIN {X 0,Y 402.157,Z 863.785,A -85,B 0,C 180,E1 -11268.73,E2 -11268.73} C_VEL
LIN {X 0,Y 403.362,Z 850.949,A -85,B 0,C 180,E1 -11269.751,E2 -11269.751} C_VEL
LIN {X 0,Y 404.343,Z 838.322,A -85,B 0,C 180,E1 -11270.541,E2 -11270.541} C_VEL
LIN {X 0,Y 405.307,Z 824.489,A -85,B 0,C 180,E1 -11271.188,E2 -11271.188} C_VEL
LIN {X 0,Y 406.022,Z 810.124,A -85,B 0,C 180,E1 -11271.648,E2 -11271.648} C_VEL
LIN {X 0,Y 407.195,Z 751.194,A -85,B 0,C 180,E1 -11272.724,E2 -11272.724} C_VEL
LIN {X 0,Y 407.85,Z 704.007,A -85,B 0,C 180,E1 -11273.578,E2 -11273.578} C_VEL
LIN {X 0,Y 403.095,Z 677.976,A -85,B 0,C 180,E1 -11274.398,E2 -11274.398} C_VEL
LIN {X 0,Y 401.716,Z 671.103,A -85,B 0,C 180,E1 -11274.635,E2 -11274.635} C_VEL
LIN {X 0,Y 402.735,Z 660.153,A -85,B 0,C 180,E1 -11276.702,E2 -11276.702} C_VEL
LIN {X 0,Y 401.048,Z 651.489,A -85,B 0,C 180,E1 -11278.538,E2 -11278.538} C_VEL
LIN {X 0,Y 398.353,Z 640.125,A -85,B 0,C 180,E1 -11281.067,E2 -11281.067} C_VEL
LIN {X 0,Y 397.096,Z 635.142,A -85,B 0,C 180,E1 -11282.22,E2 -11282.22} C_VEL
LIN {X 0,Y 397.121,Z 635.135,A -85,B 0,C 180,E1 -11285.504,E2 -11285.504} C_VEL
LIN {X 0,Y 397.136,Z 635.14,A -85,B 0,C 180,E1 -11288.863,E2 -11288.863} C_VEL
LIN {X 0,Y 397.116,Z 635.142,A -85,B 0,C 180,E1 -11292.261,E2 -11292.261} C_VEL
LIN {X 0,Y 397.089,Z 635.142,A -85,B 0,C 180,E1 -11295.069,E2 -11295.069} C_VEL
LIN {X 0,Y 397.11,Z 635.134,A -85,B 0,C 180,E1 -11298.014,E2 -11298.014} C_VEL
LIN {X 0,Y 397.138,Z 635.14,A -85,B 0,C 180,E1 -11301.137,E2 -11301.137} C_VEL
LIN {X 0,Y 397.121,Z 635.139,A -85,B 0,C 180,E1 -11304.497,E2 -11304.497} C_VEL
LIN {X 0,Y 397.078,Z 635.129,A -85,B 0,C 180,E1 -11307.929,E2 -11307.929} C_VEL
LIN {X 0,Y 397.123,Z 635.14,A -85,B 0,C 180,E1 -11311.457,E2 -11311.457} C_VEL
LIN {X 0,Y 397.153,Z 635.135,A -85,B 0,C 180,E1 -11314.488,E2 -11314.488} C_VEL
LIN {X 0,Y 397.11,Z 635.138,A -85,B 0,C 180,E1 -11317.086,E2 -11317.086} C_VEL
LIN {X 0,Y 397.149,Z 635.136,A -85,B 0,C 180,E1 -11320.353,E2 -11320.353} C_VEL
LIN {X 0,Y 397.172,Z 635.134,A -85,B 0,C 180,E1 -11323.554,E2 -11323.554} C_VEL
LIN {X 0,Y 397.229,Z 635.124,A -85,B 0,C 180,E1 -11326.703,E2 -11326.703} C_VEL
LIN {X 0,Y 397.219,Z 635.131,A -85,B 0,C 180,E1 -11329.809,E2 -11329.809} C_VEL
LIN {X 0,Y 397.352,Z 635.112,A -85,B 0,C 180,E1 -11332.888,E2 -11332.888} C_VEL
LIN {X 0,Y 397.255,Z 635.118,A -85,B 0,C 180,E1 -11334.925,E2 -11334.925} C_VEL
LIN {X 0,Y 397.45,Z 635.101,A -85,B 0,C 180,E1 -11337.974,E2 -11337.974} C_VEL
LIN {X 0,Y 397.58,Z 635.083,A -85,B 0,C 180,E1 -11340,E2 -11340} C_VEL
LIN {X 0,Y 397.377,Z 635.109,A -85,B 0,C 180,E1 -11343.042,E2 -11343.042} C_VEL
LIN {X 0,Y 397.346,Z 635.107,A -85,B 0,C 180,E1 -11346.581,E2 -11346.581} C_VEL
LIN {X 0,Y 397.254,Z 635.121,A -85,B 0,C 180,E1 -11349.162,E2 -11349.162} C_VEL
LIN {X 0,Y 397.221,Z 635.129,A -85,B 0,C 180,E1 -11352.258,E2 -11352.258} C_VEL
LIN {X 0,Y 397.182,Z 635.128,A -85,B 0,C 180,E1 -11355.392,E2 -11355.392} C_VEL
LIN {X 0,Y 397.163,Z 635.136,A -85,B 0,C 180,E1 -11358.574,E2 -11358.574} C_VEL
LIN {X 0,Y 397.098,Z 635.143,A -85,B 0,C 180,E1 -11361.819,E2 -11361.819} C_VEL
LIN {X 0,Y 397.131,Z 635.142,A -85,B 0,C 180,E1 -11365.134,E2 -11365.134} C_VEL
LIN {X 0,Y 397.081,Z 635.13,A -85,B 0,C 180,E1 -11368.547,E2 -11368.547} C_VEL
LIN {X 0,Y 397.084,Z 635.145,A -85,B 0,C 180,E1 -11371.837,E2 -11371.837} C_VEL
LIN {X 0,Y 397.127,Z 635.137,A -85,B 0,C 180,E1 -11374.494,E2 -11374.494} C_VEL
LIN {X 0,Y 397.096,Z 635.144,A -85,B 0,C 180,E1 -11378.276,E2 -11378.276} C_VEL
LIN {X 0,Y 397.056,Z 635.147,A -85,B 0,C 180,E1 -11381.977,E2 -11381.977} C_VEL
LIN {X 0,Y 397.087,Z 635.141,A -85,B 0,C 180,E1 -11385.069,E2 -11385.069} C_VEL
LIN {X 0,Y 397.055,Z 635.152,A -85,B 0,C 180,E1 -11388.024,E2 -11388.024} C_VEL
LIN {X 0,Y 397.096,Z 635.149,A -85,B 0,C 180,E1 -11391.724,E2 -11391.724} C_VEL
LIN {X 0,Y 397.12,Z 635.145,A -85,B 0,C 180,E1 -11395.506,E2 -11395.506} C_VEL
LIN {X 0,Y 397.107,Z 635.336,A -85,B 0,C 180,E1 -11397.931,E2 -11397.931} C_VEL
LIN {X 0,Y 399.21,Z 644.303,A -85,B 0,C 180,E1 -11400.247,E2 -11400.247} C_VEL
LIN {X 0,Y 406.68,Z 662.372,A -85,B 0,C 180,E1 -11401.126,E2 -11401.126} C_VEL
LIN {X 0,Y 408.384,Z 670.933,A -85,B 0,C 180,E1 -11401.406,E2 -11401.406} C_VEL
LIN {X 0,Y 406.526,Z 778.979,A -85,B 0,C 180,E1 -11403.359,E2 -11403.359} C_VEL
LIN {X 0,Y 405.923,Z 793.691,A -85,B 0,C 180,E1 -11403.801,E2 -11403.801} C_VEL
LIN {X 0,Y 405.087,Z 807.306,A -85,B 0,C 180,E1 -11404.415,E2 -11404.415} C_VEL
LIN {X 0,Y 404.118,Z 820.699,A -85,B 0,C 180,E1 -11405.236,E2 -11405.236} C_VEL
LIN {X 0,Y 402.979,Z 833.204,A -85,B 0,C 180,E1 -11406.215,E2 -11406.215} C_VEL
LIN {X 0,Y 401.825,Z 845.003,A -85,B 0,C 180,E1 -11407.37,E2 -11407.37} C_VEL
LIN {X 0,Y 400.733,Z 855.767,A -85,B 0,C 180,E1 -11408.66,E2 -11408.66} C_VEL
LIN {X 0,Y 399.51,Z 866.391,A -85,B 0,C 180,E1 -11410.206,E2 -11410.206} C_VEL
LIN {X 0,Y 398.492,Z 875.124,A -85,B 0,C 180,E1 -11411.757,E2 -11411.757} C_VEL
LIN {X 0,Y 397.642,Z 883.463,A -85,B 0,C 180,E1 -11413.573,E2 -11413.573} C_VEL
LIN {X 0,Y 396.967,Z 889.244,A -85,B 0,C 180,E1 -11415.125,E2 -11415.125} C_VEL
LIN {X 0,Y 396.532,Z 893.98,A -85,B 0,C 180,E1 -11416.679,E2 -11416.679} C_VEL
LIN {X 0,Y 396.147,Z 898.863,A -85,B 0,C 180,E1 -11418.747,E2 -11418.747} C_VEL
LIN {X 0,Y 395.87,Z 902.238,A -85,B 0,C 180,E1 -11420.806,E2 -11420.806} C_VEL
LIN {X 0,Y 395.869,Z 904.211,A -85,B 0,C 180,E1 -11422.861,E2 -11422.861} C_VEL
LIN {X 0,Y 395.798,Z 904.844,A -85,B 0,C 180,E1 -11424.907,E2 -11424.907} C_VEL
LIN {X 0,Y 395.787,Z 904.155,A -85,B 0,C 180,E1 -11426.946,E2 -11426.946} C_VEL
LIN {X 0,Y 395.861,Z 902.881,A -85,B 0,C 180,E1 -11428.341,E2 -11428.341} C_VEL
LIN {X 0,Y 395.201,Z 901.911,A -85,B 0,C 180,E1 -11429.179,E2 -11429.179} C_VEL
LIN {X 0,Y 392.475,Z 899.927,A -85,B 0,C 180,E1 -11430.536,E2 -11430.536} C_VEL
LIN {X 0,Y 390.212,Z 897.953,A -85,B 0,C 180,E1 -11431.616,E2 -11431.616} C_VEL
LIN {X 0,Y 389.277,Z 896.113,A -85,B 0,C 180,E1 -11432.433,E2 -11432.433} C_VEL
LIN {X 0,Y 389.22,Z 895.42,A -85,B 0,C 180,E1 -11432.706,E2 -11432.706} C_VEL
LIN {X 0,Y 389.761,Z 889.738,A -85,B 0,C 180,E1 -11434.654,E2 -11434.654} C_VEL
LIN {X 0,Y 390.463,Z 883.02,A -85,B 0,C 180,E1 -11436.459,E2 -11436.459} C_VEL
LIN {X 0,Y 391.066,Z 876.032,A -85,B 0,C 180,E1 -11438.006,E2 -11438.006} C_VEL
LIN {X 0,Y 391.884,Z 867.622,A -85,B 0,C 180,E1 -11439.549,E2 -11439.549} C_VEL
LIN {X 0,Y 393.142,Z 857.418,A -85,B 0,C 180,E1 -11441.08,E2 -11441.08} C_VEL
LIN {X 0,Y 394.25,Z 846.04,A -85,B 0,C 180,E1 -11442.483,E2 -11442.483} C_VEL
LIN {X 0,Y 395.362,Z 833.296,A -85,B 0,C 180,E1 -11443.754,E2 -11443.754} C_VEL
LIN {X 0,Y 396.427,Z 820.534,A -85,B 0,C 180,E1 -11444.765,E2 -11444.765} C_VEL
LIN {X 0,Y 397.365,Z 807.253,A -85,B 0,C 180,E1 -11445.582,E2 -11445.582} C_VEL
LIN {X 0,Y 398.031,Z 793.503,A -85,B 0,C 180,E1 -11446.213,E2 -11446.213} C_VEL
LIN {X 0,Y 398.521,Z 780.435,A -85,B 0,C 180,E1 -11446.62,E2 -11446.62} C_VEL
LIN {X 0,Y 400.371,Z 670.477,A -85,B 0,C 180,E1 -11448.621,E2 -11448.621} C_VEL
LIN {X 0,Y 397.812,Z 659.838,A -85,B 0,C 180,E1 -11448.975,E2 -11448.975} C_VEL
LIN {X 0,Y 391.875,Z 644.279,A -85,B 0,C 180,E1 -11449.654,E2 -11449.654} C_VEL
LIN {X 0,Y 390.078,Z 636.023,A -85,B 0,C 180,E1 -11451.745,E2 -11451.745} C_VEL
LIN {X 0,Y 390.045,Z 636.028,A -85,B 0,C 180,E1 -11454.483,E2 -11454.483} C_VEL
LIN {X 0,Y 390.018,Z 636.029,A -85,B 0,C 180,E1 -11457.997,E2 -11457.997} C_VEL
LIN {X 0,Y 390.02,Z 636.027,A -85,B 0,C 180,E1 -11461.505,E2 -11461.505} C_VEL
LIN {X 0,Y 390.071,Z 636.022,A -85,B 0,C 180,E1 -11465.209,E2 -11465.209} C_VEL
LIN {X 0,Y 390.06,Z 636.012,A -85,B 0,C 180,E1 -11469.096,E2 -11469.096} C_VEL
LIN {X 0,Y 390.033,Z 636.024,A -85,B 0,C 180,E1 -11472.372,E2 -11472.372} C_VEL
LIN {X 0,Y 390.044,Z 636.025,A -85,B 0,C 180,E1 -11475.354,E2 -11475.354} C_VEL
LIN {X 0,Y 390.017,Z 636.024,A -85,B 0,C 180,E1 -11478.184,E2 -11478.184} C_VEL
LIN {X 0,Y 390.06,Z 636.015,A -85,B 0,C 180,E1 -11480.903,E2 -11480.903} C_VEL
LIN {X 0,Y 390.075,Z 636.01,A -85,B 0,C 180,E1 -11484.792,E2 -11484.792} C_VEL
LIN {X 0,Y 390.026,Z 636.022,A -85,B 0,C 180,E1 -11488.495,E2 -11488.495} C_VEL
LIN {X 0,Y 390.031,Z 636.023,A -85,B 0,C 180,E1 -11492.063,E2 -11492.063} C_VEL
LIN {X 0,Y 390.045,Z 636.014,A -85,B 0,C 180,E1 -11495.517,E2 -11495.517} C_VEL
LIN {X 0,Y 390.058,Z 636.02,A -85,B 0,C 180,E1 -11498.877,E2 -11498.877} C_VEL
LIN {X 0,Y 390.114,Z 636,A -85,B 0,C 180,E1 -11502.166,E2 -11502.166} C_VEL
LIN {X 0,Y 390.147,Z 636.011,A -85,B 0,C 180,E1 -11505.392,E2 -11505.392} C_VEL
LIN {X 0,Y 390.15,Z 636,A -85,B 0,C 180,E1 -11508.571,E2 -11508.571} C_VEL
LIN {X 0,Y 390.259,Z 635.996,A -85,B 0,C 180,E1 -11512.086,E2 -11512.086} C_VEL
LIN {X 0,Y 390.215,Z 635.998,A -85,B 0,C 180,E1 -11514.833,E2 -11514.833} C_VEL
LIN {X 0,Y 390.418,Z 635.98,A -85,B 0,C 180,E1 -11517.936,E2 -11517.936} C_VEL
LIN {X 0,Y 390.549,Z 635.957,A -85,B 0,C 180,E1 -11520,E2 -11520} C_VEL
LIN {X 0,Y 390.311,Z 635.988,A -85,B 0,C 180,E1 -11523.096,E2 -11523.096} C_VEL
LIN {X 0,Y 390.306,Z 635.989,A -85,B 0,C 180,E1 -11526.202,E2 -11526.202} C_VEL
LIN {X 0,Y 390.279,Z 635.995,A -85,B 0,C 180,E1 -11528.283,E2 -11528.283} C_VEL
LIN {X 0,Y 390.15,Z 636.004,A -85,B 0,C 180,E1 -11531.429,E2 -11531.429} C_VEL
LIN {X 0,Y 390.149,Z 636.004,A -85,B 0,C 180,E1 -11534.607,E2 -11534.607} C_VEL
LIN {X 0,Y 390.131,Z 636.013,A -85,B 0,C 180,E1 -11537.833,E2 -11537.833} C_VEL
LIN {X 0,Y 390.057,Z 636.017,A -85,B 0,C 180,E1 -11541.122,E2 -11541.122} C_VEL
LIN {X 0,Y 390.079,Z 636.019,A -85,B 0,C 180,E1 -11544.481,E2 -11544.481} C_VEL
LIN {X 0,Y 390.119,Z 636.01,A -85,B 0,C 180,E1 -11547.93,E2 -11547.93} C_VEL
LIN {X 0,Y 390.025,Z 636.022,A -85,B 0,C 180,E1 -11551.504,E2 -11551.504} C_VEL
LIN {X 0,Y 390.07,Z 636.02,A -85,B 0,C 180,E1 -11554.024,E2 -11554.024} C_VEL
LIN {X 0,Y 390.048,Z 636.02,A -85,B 0,C 180,E1 -11557.551,E2 -11557.551} C_VEL
LIN {X 0,Y 390.078,Z 636.02,A -85,B 0,C 180,E1 -11560.825,E2 -11560.825} C_VEL
LIN {X 0,Y 390.057,Z 636.02,A -85,B 0,C 180,E1 -11563.886,E2 -11563.886} C_VEL
LIN {X 0,Y 390.06,Z 636.016,A -85,B 0,C 180,E1 -11566.79,E2 -11566.79} C_VEL
LIN {X 0,Y 390.059,Z 636.021,A -85,B 0,C 180,E1 -11569.561,E2 -11569.561} C_VEL
LIN {X 0,Y 390.047,Z 636.026,A -85,B 0,C 180,E1 -11572.448,E2 -11572.448} C_VEL
LIN {X 0,Y 390.085,Z 636.019,A -85,B 0,C 180,E1 -11576.047,E2 -11576.047} C_VEL
LIN {X 0,Y 390.053,Z 636.092,A -85,B 0,C 180,E1 -11578.333,E2 -11578.333} C_VEL
LIN {X 0,Y 393.345,Z 650.016,A -85,B 0,C 180,E1 -11581.369,E2 -11581.369} C_VEL
LIN {X 0,Y 395.174,Z 659.482,A -85,B 0,C 180,E1 -11583.339,E2 -11583.339} C_VEL
LIN {X 0,Y 394.193,Z 671.015,A -85,B 0,C 180,E1 -11585.51,E2 -11585.51} C_VEL
LIN {X 0,Y 400.023,Z 705.507,A -85,B 0,C 180,E1 -11586.519,E2 -11586.519} C_VEL
LIN {X 0,Y 398.278,Z 808.458,A -85,B 0,C 180,E1 -11588.385,E2 -11588.385} C_VEL
LIN {X 0,Y 397.664,Z 822.783,A -85,B 0,C 180,E1 -11588.826,E2 -11588.826} C_VEL
LIN {X 0,Y 396.78,Z 836.58,A -85,B 0,C 180,E1 -11589.456,E2 -11589.456} C_VEL
LIN {X 0,Y 395.798,Z 849.957,A -85,B 0,C 180,E1 -11590.283,E2 -11590.283} C_VEL
LIN {X 0,Y 394.656,Z 862.837,A -85,B 0,C 180,E1 -11591.304,E2 -11591.304} C_VEL
LIN {X 0,Y 393.468,Z 874.545,A -85,B 0,C 180,E1 -11592.457,E2 -11592.457} C_VEL
LIN {X 0,Y 392.282,Z 886.261,A -85,B 0,C 180,E1 -11593.877,E2 -11593.877} C_VEL
LIN {X 0,Y 391.178,Z 896.732,A -85,B 0,C 180,E1 -11595.432,E2 -11595.432} C_VEL
LIN {X 0,Y 390.493,Z 905.381,A -85,B 0,C 180,E1 -11596.999,E2 -11596.999} C_VEL
LIN {X 0,Y 389.699,Z 913.632,A -85,B 0,C 180,E1 -11598.821,E2 -11598.821} C_VEL
LIN {X 0,Y 389.18,Z 920.278,A -85,B 0,C 180,E1 -11600.646,E2 -11600.646} C_VEL
LIN {X 0,Y 388.846,Z 926.173,A -85,B 0,C 180,E1 -11602.731,E2 -11602.731} C_VEL
LIN {X 0,Y 388.833,Z 928.517,A -85,B 0,C 180,E1 -11603.774,E2 -11603.774} C_VEL
LIN {X 0,Y 388.691,Z 932.073,A -85,B 0,C 180,E1 -11605.852,E2 -11605.852} C_VEL
LIN {X 0,Y 388.714,Z 934.22,A -85,B 0,C 180,E1 -11607.928,E2 -11607.928} C_VEL
LIN {X 0,Y 388.724,Z 935.007,A -85,B 0,C 180,E1 -11610,E2 -11610} C_VEL
LIN {X 0,Y 388.695,Z 934.453,A -85,B 0,C 180,E1 -11612.072,E2 -11612.072} C_VEL
LIN {X 0,Y 388.691,Z 932.556,A -85,B 0,C 180,E1 -11614.147,E2 -11614.147} C_VEL
LIN {X 0,Y 388.804,Z 929.26,A -85,B 0,C 180,E1 -11616.226,E2 -11616.226} C_VEL
LIN {X 0,Y 388.997,Z 924.462,A -85,B 0,C 180,E1 -11618.31,E2 -11618.31} C_VEL
LIN {X 0,Y 389.332,Z 919.84,A -85,B 0,C 180,E1 -11619.874,E2 -11619.874} C_VEL
LIN {X 0,Y 389.985,Z 913.15,A -85,B 0,C 180,E1 -11621.697,E2 -11621.697} C_VEL
LIN {X 0,Y 390.866,Z 904.841,A -85,B 0,C 180,E1 -11623.518,E2 -11623.518} C_VEL
LIN {X 0,Y 391.718,Z 896.196,A -85,B 0,C 180,E1 -11625.079,E2 -11625.079} C_VEL
LIN {X 0,Y 392.928,Z 885.743,A -85,B 0,C 180,E1 -11626.629,E2 -11626.629} C_VEL
LIN {X 0,Y 394.148,Z 875.246,A -85,B 0,C 180,E1 -11627.914,E2 -11627.914} C_VEL
LIN {X 0,Y 395.442,Z 863.843,A -85,B 0,C 180,E1 -11629.061,E2 -11629.061} C_VEL
LIN {X 0,Y 396.692,Z 850.793,A -85,B 0,C 180,E1 -11630.12,E2 -11630.12} C_VEL
LIN {X 0,Y 397.827,Z 837.452,A -85,B 0,C 180,E1 -11630.961,E2 -11630.961} C_VEL
LIN {X 0,Y 398.783,Z 823.417,A -85,B 0,C 180,E1 -11631.62,E2 -11631.62} C_VEL
LIN {X 0,Y 399.565,Z 808.593,A -85,B 0,C 180,E1 -11632.084,E2 -11632.084} C_VEL
LIN {X 0,Y 401.503,Z 705.657,A -85,B 0,C 180,E1 -11633.97,E2 -11633.97} C_VEL
LIN {X 0,Y 397.138,Z 681.305,A -85,B 0,C 180,E1 -11634.75,E2 -11634.75} C_VEL
LIN {X 0,Y 394.987,Z 670.848,A -85,B 0,C 180,E1 -11635.114,E2 -11635.114} C_VEL
LIN {X 0,Y 395.918,Z 661.802,A -85,B 0,C 180,E1 -11636.851,E2 -11636.851} C_VEL
LIN {X 0,Y 393.903,Z 651.709,A -85,B 0,C 180,E1 -11639.043,E2 -11639.043} C_VEL
LIN {X 0,Y 391.09,Z 640.198,A -85,B 0,C 180,E1 -11641.682,E2 -11641.682} C_VEL
LIN {X 0,Y 390.07,Z 636.014,A -85,B 0,C 180,E1 -11642.719,E2 -11642.719} C_VEL
LIN {X 0,Y 390.058,Z 636.017,A -85,B 0,C 180,E1 -11645.826,E2 -11645.826} C_VEL
LIN {X 0,Y 390.074,Z 636.023,A -85,B 0,C 180,E1 -11649.219,E2 -11649.219} C_VEL
LIN {X 0,Y 390.082,Z 636.018,A -85,B 0,C 180,E1 -11652.381,E2 -11652.381} C_VEL
LIN {X 0,Y 390.056,Z 636.021,A -85,B 0,C 180,E1 -11656.114,E2 -11656.114} C_VEL
LIN {X 0,Y 390.076,Z 636.019,A -85,B 0,C 180,E1 -11659.563,E2 -11659.563} C_VEL
LIN {X 0,Y 390.048,Z 636.007,A -85,B 0,C 180,E1 -11662.449,E2 -11662.449} C_VEL
LIN {X 0,Y 390.084,Z 636.017,A -85,B 0,C 180,E1 -11666.047,E2 -11666.047} C_VEL
LIN {X 0,Y 390.047,Z 636.01,A -85,B 0,C 180,E1 -11669.869,E2 -11669.869} C_VEL
LIN {X 0,Y 390.114,Z 636.011,A -85,B 0,C 180,E1 -11673.232,E2 -11673.232} C_VEL
LIN {X 0,Y 390.107,Z 636.01,A -85,B 0,C 180,E1 -11676.75,E2 -11676.75} C_VEL
LIN {X 0,Y 390.105,Z 636.018,A -85,B 0,C 180,E1 -11679.983,E2 -11679.983} C_VEL
LIN {X 0,Y 390.142,Z 636.008,A -85,B 0,C 180,E1 -11683.249,E2 -11683.249} C_VEL
LIN {X 0,Y 390.195,Z 636.001,A -85,B 0,C 180,E1 -11686.562,E2 -11686.562} C_VEL
LIN {X 0,Y 390.17,Z 636.007,A -85,B 0,C 180,E1 -11689.623,E2 -11689.623} C_VEL
LIN {X 0,Y 390.303,Z 635.991,A -85,B 0,C 180,E1 -11692.759,E2 -11692.759} C_VEL
LIN {X 0,Y 390.227,Z 635.994,A -85,B 0,C 180,E1 -11694.834,E2 -11694.834} C_VEL
LIN {X 0,Y 390.419,Z 635.977,A -85,B 0,C 180,E1 -11697.937,E2 -11697.937} C_VEL
LIN {X 0,Y 390.55,Z 635.958,A -85,B 0,C 180,E1 -11700,E2 -11700} C_VEL
LIN {X 0,Y 390.312,Z 635.989,A -85,B 0,C 180,E1 -11703.097,E2 -11703.097} C_VEL
LIN {X 0,Y 390.303,Z 635.984,A -85,B 0,C 180,E1 -11706.575,E2 -11706.575} C_VEL
LIN {X 0,Y 390.206,Z 635.998,A -85,B 0,C 180,E1 -11709.329,E2 -11709.329} C_VEL
LIN {X 0,Y 390.196,Z 636.002,A -85,B 0,C 180,E1 -11713.439,E2 -11713.439} C_VEL
LIN {X 0,Y 390.151,Z 636.009,A -85,B 0,C 180,E1 -11717.308,E2 -11717.308} C_VEL
LIN {X 0,Y 390.089,Z 636.015,A -85,B 0,C 180,E1 -11720.47,E2 -11720.47} C_VEL
LIN {X 0,Y 390.068,Z 636.014,A -85,B 0,C 180,E1 -11723.353,E2 -11723.353} C_VEL
LIN {X 0,Y 390.058,Z 636.019,A -85,B 0,C 180,E1 -11726.773,E2 -11726.773} C_VEL
LIN {X 0,Y 390.039,Z 636.01,A -85,B 0,C 180,E1 -11730.3,E2 -11730.3} C_VEL
LIN {X 0,Y 390.07,Z 636.014,A -85,B 0,C 180,E1 -11734.025,E2 -11734.025} C_VEL
LIN {X 0,Y 390.042,Z 636.024,A -85,B 0,C 180,E1 -11737.55,E2 -11737.55} C_VEL
LIN {X 0,Y 390.02,Z 636.016,A -85,B 0,C 180,E1 -11740.815,E2 -11740.815} C_VEL
LIN {X 0,Y 390.054,Z 636.022,A -85,B 0,C 180,E1 -11743.886,E2 -11743.886} C_VEL
LIN {X 0,Y 390.049,Z 636.024,A -85,B 0,C 180,E1 -11746.789,E2 -11746.789} C_VEL
LIN {X 0,Y 390.012,Z 636.032,A -85,B 0,C 180,E1 -11749.555,E2 -11749.555} C_VEL
LIN {X 0,Y 390.043,Z 636.026,A -85,B 0,C 180,E1 -11752.45,E2 -11752.45} C_VEL
LIN {X 0,Y 390.064,Z 636.019,A -85,B 0,C 180,E1 -11756.045,E2 -11756.045} C_VEL
LIN {X 0,Y 390.089,Z 636.177,A -85,B 0,C 180,E1 -11757.497,E2 -11757.497} C_VEL
LIN {X 0,Y 392.147,Z 644.84,A -85,B 0,C 180,E1 -11759.735,E2 -11759.735} C_VEL
LIN {X 0,Y 400.528,Z 664.619,A -85,B 0,C 180,E1 -11760.742,E2 -11760.742} C_VEL
LIN {X 0,Y 402,Z 671.782,A -85,B 0,C 180,E1 -11760.985,E2 -11760.985} C_VEL
LIN {X 0,Y 400.015,Z 780.904,A -85,B 0,C 180,E1 -11762.996,E2 -11762.996} C_VEL
LIN {X 0,Y 399.308,Z 795.641,A -85,B 0,C 180,E1 -11763.474,E2 -11763.474} C_VEL
LIN {X 0,Y 398.341,Z 809.511,A -85,B 0,C 180,E1 -11764.133,E2 -11764.133} C_VEL
LIN {X 0,Y 397.326,Z 823.169,A -85,B 0,C 180,E1 -11765.02,E2 -11765.02} C_VEL
LIN {X 0,Y 396.124,Z 835.69,A -85,B 0,C 180,E1 -11766.056,E2 -11766.056} C_VEL
LIN {X 0,Y 394.916,Z 847.331,A -85,B 0,C 180,E1 -11767.256,E2 -11767.256} C_VEL
LIN {X 0,Y 393.767,Z 857.749,A -85,B 0,C 180,E1 -11768.566,E2 -11768.566} C_VEL
LIN {X 0,Y 392.538,Z 867.902,A -85,B 0,C 180,E1 -11770.112,E2 -11770.112} C_VEL
LIN {X 0,Y 391.488,Z 876.422,A -85,B 0,C 180,E1 -11771.69,E2 -11771.69} C_VEL
LIN {X 0,Y 390.593,Z 884.516,A -85,B 0,C 180,E1 -11773.537,E2 -11773.537} C_VEL
LIN {X 0,Y 389.823,Z 891.011,A -85,B 0,C 180,E1 -11775.38,E2 -11775.38} C_VEL
LIN {X 0,Y 389.282,Z 896.747,A -85,B 0,C 180,E1 -11777.488,E2 -11777.488} C_VEL
LIN {X 0,Y 388.888,Z 900.901,A -85,B 0,C 180,E1 -11779.588,E2 -11779.588} C_VEL
LIN {X 0,Y 388.773,Z 903.603,A -85,B 0,C 180,E1 -11781.685,E2 -11781.685} C_VEL
LIN {X 0,Y 388.778,Z 904.942,A -85,B 0,C 180,E1 -11783.773,E2 -11783.773} C_VEL
LIN {X 0,Y 388.682,Z 904.961,A -85,B 0,C 180,E1 -11785.852,E2 -11785.852} C_VEL
LIN {X 0,Y 388.799,Z 903.652,A -85,B 0,C 180,E1 -11787.928,E2 -11787.928} C_VEL
LIN {X 0,Y 388.794,Z 901.012,A -85,B 0,C 180,E1 -11790,E2 -11790} C_VEL
LIN {X 0,Y 389.018,Z 896.962,A -85,B 0,C 180,E1 -11792.071,E2 -11792.071} C_VEL
LIN {X 0,Y 389.22,Z 895.42,A -85,B 0,C 180,E1 -11792.706,E2 -11792.706} C_VEL
LIN {X 0,Y 388.649,Z 893.316,A -85,B 0,C 180,E1 -11793.515,E2 -11793.515} C_VEL
LIN {X 0,Y 386.076,Z 889.56,A -85,B 0,C 180,E1 -11794.826,E2 -11794.826} C_VEL
LIN {X 0,Y 383.728,Z 885.304,A -85,B 0,C 180,E1 -11796.114,E2 -11796.114} C_VEL
LIN {X 0,Y 383.505,Z 882.312,A -85,B 0,C 180,E1 -11796.875,E2 -11796.875} C_VEL
LIN {X 0,Y 384.061,Z 876.599,A -85,B 0,C 180,E1 -11798.153,E2 -11798.153} C_VEL
LIN {X 0,Y 384.922,Z 868.243,A -85,B 0,C 180,E1 -11799.723,E2 -11799.723} C_VEL
LIN {X 0,Y 386.208,Z 858.137,A -85,B 0,C 180,E1 -11801.281,E2 -11801.281} C_VEL
LIN {X 0,Y 387.367,Z 846.847,A -85,B 0,C 180,E1 -11802.708,E2 -11802.708} C_VEL
LIN {X 0,Y 388.424,Z 835.621,A -85,B 0,C 180,E1 -11803.871,E2 -11803.871} C_VEL
LIN {X 0,Y 389.541,Z 823.342,A -85,B 0,C 180,E1 -11804.898,E2 -11804.898} C_VEL
LIN {X 0,Y 390.468,Z 810.778,A -85,B 0,C 180,E1 -11805.73,E2 -11805.73} C_VEL
LIN {X 0,Y 391.229,Z 796.689,A -85,B 0,C 180,E1 -11806.435,E2 -11806.435} C_VEL
LIN {X 0,Y 391.792,Z 782.789,A -85,B 0,C 180,E1 -11806.914,E2 -11806.914} C_VEL
LIN {X 0,Y 392.252,Z 758.779,A -85,B 0,C 180,E1 -11807.397,E2 -11807.397} C_VEL
LIN {X 0,Y 393.777,Z 671.517,A -85,B 0,C 180,E1 -11808.991,E2 -11808.991} C_VEL
LIN {X 0,Y 391.519,Z 662.172,A -85,B 0,C 180,E1 -11809.31,E2 -11809.31} C_VEL
LIN {X 0,Y 384.738,Z 644.582,A -85,B 0,C 180,E1 -11810.098,E2 -11810.098} C_VEL
LIN {X 0,Y 383.022,Z 636.902,A -85,B 0,C 180,E1 -11812.096,E2 -11812.096} C_VEL
LIN {X 0,Y 382.989,Z 636.906,A -85,B 0,C 180,E1 -11814.965,E2 -11814.965} C_VEL
LIN {X 0,Y 382.978,Z 636.904,A -85,B 0,C 180,E1 -11818.498,E2 -11818.498} C_VEL
LIN {X 0,Y 383.006,Z 636.901,A -85,B 0,C 180,E1 -11822.15,E2 -11822.15} C_VEL
LIN {X 0,Y 383.014,Z 636.901,A -85,B 0,C 180,E1 -11824.669,E2 -11824.669} C_VEL
LIN {X 0,Y 382.995,Z 636.9,A -85,B 0,C 180,E1 -11827.902,E2 -11827.902} C_VEL
LIN {X 0,Y 382.963,Z 636.906,A -85,B 0,C 180,E1 -11831.35,E2 -11831.35} C_VEL
LIN {X 0,Y 382.992,Z 636.897,A -85,B 0,C 180,E1 -11834.302,E2 -11834.302} C_VEL
LIN {X 0,Y 382.999,Z 636.9,A -85,B 0,C 180,E1 -11837.238,E2 -11837.238} C_VEL
LIN {X 0,Y 382.988,Z 636.899,A -85,B 0,C 180,E1 -11840.419,E2 -11840.419} C_VEL
LIN {X 0,Y 383.018,Z 636.886,A -85,B 0,C 180,E1 -11844.043,E2 -11844.043} C_VEL
LIN {X 0,Y 382.99,Z 636.901,A -85,B 0,C 180,E1 -11847.578,E2 -11847.578} C_VEL
LIN {X 0,Y 382.981,Z 636.893,A -85,B 0,C 180,E1 -11850.299,E2 -11850.299} C_VEL
LIN {X 0,Y 383.006,Z 636.896,A -85,B 0,C 180,E1 -11854.044,E2 -11854.044} C_VEL
LIN {X 0,Y 382.992,Z 636.897,A -85,B 0,C 180,E1 -11857.334,E2 -11857.334} C_VEL
LIN {X 0,Y 383.062,Z 636.889,A -85,B 0,C 180,E1 -11860.716,E2 -11860.716} C_VEL
LIN {X 0,Y 383.084,Z 636.887,A -85,B 0,C 180,E1 -11864.026,E2 -11864.026} C_VEL
LIN {X 0,Y 383.139,Z 636.884,A -85,B 0,C 180,E1 -11867.284,E2 -11867.284} C_VEL
LIN {X 0,Y 383.146,Z 636.872,A -85,B 0,C 180,E1 -11870.497,E2 -11870.497} C_VEL
LIN {X 0,Y 383.245,Z 636.874,A -85,B 0,C 180,E1 -11873.683,E2 -11873.683} C_VEL
LIN {X 0,Y 383.386,Z 636.856,A -85,B 0,C 180,E1 -11877.899,E2 -11877.899} C_VEL
LIN {X 0,Y 383.518,Z 636.833,A -85,B 0,C 180,E1 -11880,E2 -11880} C_VEL
LIN {X 0,Y 383.248,Z 636.868,A -85,B 0,C 180,E1 -11883.153,E2 -11883.153} C_VEL
LIN {X 0,Y 383.263,Z 636.866,A -85,B 0,C 180,E1 -11886.316,E2 -11886.316} C_VEL
LIN {X 0,Y 383.224,Z 636.872,A -85,B 0,C 180,E1 -11888.436,E2 -11888.436} C_VEL
LIN {X 0,Y 383.099,Z 636.884,A -85,B 0,C 180,E1 -11891.642,E2 -11891.642} C_VEL
LIN {X 0,Y 383.115,Z 636.879,A -85,B 0,C 180,E1 -11894.881,E2 -11894.881} C_VEL
LIN {X 0,Y 383.092,Z 636.889,A -85,B 0,C 180,E1 -11898.172,E2 -11898.172} C_VEL
LIN {X 0,Y 382.994,Z 636.898,A -85,B 0,C 180,E1 -11901.531,E2 -11901.531} C_VEL
LIN {X 0,Y 383.052,Z 636.891,A -85,B 0,C 180,E1 -11904.96,E2 -11904.96} C_VEL
LIN {X 0,Y 383.042,Z 636.898,A -85,B 0,C 180,E1 -11908.492,E2 -11908.492} C_VEL
LIN {X 0,Y 383.011,Z 636.9,A -85,B 0,C 180,E1 -11912.149,E2 -11912.149} C_VEL
LIN {X 0,Y 383.019,Z 636.901,A -85,B 0,C 180,E1 -11914.668,E2 -11914.668} C_VEL
LIN {X 0,Y 383.004,Z 636.9,A -85,B 0,C 180,E1 -11917.904,E2 -11917.904} C_VEL
LIN {X 0,Y 383.015,Z 636.896,A -85,B 0,C 180,E1 -11921.343,E2 -11921.343} C_VEL
LIN {X 0,Y 382.998,Z 636.901,A -85,B 0,C 180,E1 -11924.303,E2 -11924.303} C_VEL
LIN {X 0,Y 383.011,Z 636.896,A -85,B 0,C 180,E1 -11927.24,E2 -11927.24} C_VEL
LIN {X 0,Y 383.018,Z 636.901,A -85,B 0,C 180,E1 -11930.413,E2 -11930.413} C_VEL
LIN {X 0,Y 383.028,Z 636.899,A -85,B 0,C 180,E1 -11934.045,E2 -11934.045} C_VEL
LIN {X 0,Y 382.988,Z 636.903,A -85,B 0,C 180,E1 -11937.578,E2 -11937.578} C_VEL
LIN {X 0,Y 383.012,Z 636.952,A -85,B 0,C 180,E1 -11937.967,E2 -11937.967} C_VEL
LIN {X 0,Y 386.559,Z 651.965,A -85,B 0,C 180,E1 -11941.305,E2 -11941.305} C_VEL
LIN {X 0,Y 388.219,Z 660.357,A -85,B 0,C 180,E1 -11943.091,E2 -11943.091} C_VEL
LIN {X 0,Y 387.41,Z 670.803,A -85,B 0,C 180,E1 -11945.101,E2 -11945.101} C_VEL
LIN {X 0,Y 393.436,Z 706.203,A -85,B 0,C 180,E1 -11946.154,E2 -11946.154} C_VEL
LIN {X 0,Y 391.619,Z 808.244,A -85,B 0,C 180,E1 -11948.033,E2 -11948.033} C_VEL
LIN {X 0,Y 390.982,Z 822.543,A -85,B 0,C 180,E1 -11948.481,E2 -11948.481} C_VEL
LIN {X 0,Y 390.091,Z 835.759,A -85,B 0,C 180,E1 -11949.087,E2 -11949.087} C_VEL
LIN {X 0,Y 389.027,Z 849.614,A -85,B 0,C 180,E1 -11949.953,E2 -11949.953} C_VEL
LIN {X 0,Y 387.884,Z 862.223,A -85,B 0,C 180,E1 -11950.965,E2 -11950.965} C_VEL
LIN {X 0,Y 386.648,Z 873.992,A -85,B 0,C 180,E1 -11952.137,E2 -11952.137} C_VEL
LIN {X 0,Y 385.628,Z 883.786,A -85,B 0,C 180,E1 -11953.319,E2 -11953.319} C_VEL
LIN {X 0,Y 384.419,Z 894.624,A -85,B 0,C 180,E1 -11954.899,E2 -11954.899} C_VEL
LIN {X 0,Y 383.611,Z 903.579,A -85,B 0,C 180,E1 -11956.491,E2 -11956.491} C_VEL
LIN {X 0,Y 382.772,Z 912.149,A -85,B 0,C 180,E1 -11958.348,E2 -11958.348} C_VEL
LIN {X 0,Y 382.235,Z 918.133,A -85,B 0,C 180,E1 -11959.94,E2 -11959.94} C_VEL
LIN {X 0,Y 381.931,Z 923.08,A -85,B 0,C 180,E1 -11961.535,E2 -11961.535} C_VEL
LIN {X 0,Y 381.738,Z 928.182,A -85,B 0,C 180,E1 -11963.658,E2 -11963.658} C_VEL
LIN {X 0,Y 381.617,Z 931.76,A -85,B 0,C 180,E1 -11965.775,E2 -11965.775} C_VEL
LIN {X 0,Y 381.613,Z 933.924,A -85,B 0,C 180,E1 -11967.889,E2 -11967.889} C_VEL
LIN {X 0,Y 381.654,Z 934.731,A -85,B 0,C 180,E1 -11970,E2 -11970} C_VEL
LIN {X 0,Y 381.594,Z 934.192,A -85,B 0,C 180,E1 -11972.111,E2 -11972.111} C_VEL
LIN {X 0,Y 381.616,Z 932.315,A -85,B 0,C 180,E1 -11974.224,E2 -11974.224} C_VEL
LIN {X 0,Y 381.711,Z 929.043,A -85,B 0,C 180,E1 -11976.342,E2 -11976.342} C_VEL
LIN {X 0,Y 381.945,Z 924.268,A -85,B 0,C 180,E1 -11978.465,E2 -11978.465} C_VEL
LIN {X 0,Y 382.412,Z 917.871,A -85,B 0,C 180,E1 -11980.59,E2 -11980.59} C_VEL
LIN {X 0,Y 383.239,Z 910.773,A -85,B 0,C 180,E1 -11982.443,E2 -11982.443} C_VEL
LIN {X 0,Y 384.181,Z 901.957,A -85,B 0,C 180,E1 -11984.307,E2 -11984.307} C_VEL
LIN {X 0,Y 385.202,Z 892.851,A -85,B 0,C 180,E1 -11985.883,E2 -11985.883} C_VEL
LIN {X 0,Y 386.565,Z 881.779,A -85,B 0,C 180,E1 -11987.456,E2 -11987.456} C_VEL
LIN {X 0,Y 387.987,Z 870.504,A -85,B 0,C 180,E1 -11988.755,E2 -11988.755} C_VEL
LIN {X 0,Y 389.315,Z 858.062,A -85,B 0,C 180,E1 -11989.922,E2 -11989.922} C_VEL
LIN {X 0,Y 390.469,Z 846.032,A -85,B 0,C 180,E1 -11990.826,E2 -11990.826} C_VEL
LIN {X 0,Y 391.571,Z 832.967,A -85,B 0,C 180,E1 -11991.588,E2 -11991.588} C_VEL
LIN {X 0,Y 392.571,Z 818.814,A -85,B 0,C 180,E1 -11992.187,E2 -11992.187} C_VEL
LIN {X 0,Y 393.166,Z 803.821,A -85,B 0,C 180,E1 -11992.602,E2 -11992.602} C_VEL
LIN {X 0,Y 395.063,Z 707.207,A -85,B 0,C 180,E1 -11994.384,E2 -11994.384} C_VEL
LIN {X 0,Y 392.187,Z 689.769,A -85,B 0,C 180,E1 -11994.937,E2 -11994.937} C_VEL
LIN {X 0,Y 388.304,Z 670.416,A -85,B 0,C 180,E1 -11995.646,E2 -11995.646} C_VEL
LIN {X 0,Y 389.028,Z 662.927,A -85,B 0,C 180,E1 -11997.117,E2 -11997.117} C_VEL
LIN {X 0,Y 386.321,Z 649.974,A -85,B 0,C 180,E1 -12000.019,E2 -12000.019} C_VEL
LIN {X 0,Y 383.036,Z 636.888,A -85,B 0,C 180,E1 -12003.145,E2 -12003.145} C_VEL
LIN {X 0,Y 383.034,Z 636.894,A -85,B 0,C 180,E1 -12006.165,E2 -12006.165} C_VEL
LIN {X 0,Y 383.019,Z 636.894,A -85,B 0,C 180,E1 -12009.957,E2 -12009.957} C_VEL
LIN {X 0,Y 383.032,Z 636.897,A -85,B 0,C 180,E1 -12012.783,E2 -12012.783} C_VEL
LIN {X 0,Y 382.999,Z 636.902,A -85,B 0,C 180,E1 -12015.79,E2 -12015.79} C_VEL
LIN {X 0,Y 383.016,Z 636.892,A -85,B 0,C 180,E1 -12018.791,E2 -12018.791} C_VEL
LIN {X 0,Y 383.004,Z 636.886,A -85,B 0,C 180,E1 -12022.096,E2 -12022.096} C_VEL
LIN {X 0,Y 383.019,Z 636.899,A -85,B 0,C 180,E1 -12025.332,E2 -12025.332} C_VEL
LIN {X 0,Y 382.983,Z 636.881,A -85,B 0,C 180,E1 -12029.082,E2 -12029.082} C_VEL
LIN {X 0,Y 383.057,Z 636.889,A -85,B 0,C 180,E1 -12032.698,E2 -12032.698} C_VEL
LIN {X 0,Y 383.034,Z 636.895,A -85,B 0,C 180,E1 -12036.193,E2 -12036.193} C_VEL
LIN {X 0,Y 383.056,Z 636.894,A -85,B 0,C 180,E1 -12039.599,E2 -12039.599} C_VEL
LIN {X 0,Y 383.108,Z 636.884,A -85,B 0,C 180,E1 -12042.932,E2 -12042.932} C_VEL
LIN {X 0,Y 383.126,Z 636.881,A -85,B 0,C 180,E1 -12046.464,E2 -12046.464} C_VEL
LIN {X 0,Y 383.153,Z 636.875,A -85,B 0,C 180,E1 -12050.498,E2 -12050.498} C_VEL
LIN {X 0,Y 383.282,Z 636.866,A -85,B 0,C 180,E1 -12053.684,E2 -12053.684} C_VEL
LIN {X 0,Y 383.387,Z 636.852,A -85,B 0,C 180,E1 -12057.899,E2 -12057.899} C_VEL
LIN {X 0,Y 383.519,Z 636.833,A -85,B 0,C 180,E1 -12060,E2 -12060} C_VEL
LIN {X 0,Y 383.248,Z 636.869,A -85,B 0,C 180,E1 -12063.154,E2 -12063.154} C_VEL
LIN {X 0,Y 383.264,Z 636.862,A -85,B 0,C 180,E1 -12066.566,E2 -12066.566} C_VEL
LIN {X 0,Y 383.153,Z 636.877,A -85,B 0,C 180,E1 -12069.502,E2 -12069.502} C_VEL
LIN {X 0,Y 383.127,Z 636.882,A -85,B 0,C 180,E1 -12073.536,E2 -12073.536} C_VEL
LIN {X 0,Y 383.096,Z 636.887,A -85,B 0,C 180,E1 -12077.455,E2 -12077.455} C_VEL
LIN {X 0,Y 383.031,Z 636.896,A -85,B 0,C 180,E1 -12080.647,E2 -12080.647} C_VEL
LIN {X 0,Y 383.02,Z 636.891,A -85,B 0,C 180,E1 -12083.809,E2 -12083.809} C_VEL
LIN {X 0,Y 382.996,Z 636.892,A -85,B 0,C 180,E1 -12087.307,E2 -12087.307} C_VEL
LIN {X 0,Y 382.984,Z 636.895,A -85,B 0,C 180,E1 -12090.919,E2 -12090.919} C_VEL
LIN {X 0,Y 383.02,Z 636.896,A -85,B 0,C 180,E1 -12094.668,E2 -12094.668} C_VEL
LIN {X 0,Y 382.996,Z 636.901,A -85,B 0,C 180,E1 -12097.903,E2 -12097.903} C_VEL
LIN {X 0,Y 382.963,Z 636.896,A -85,B 0,C 180,E1 -12101.351,E2 -12101.351} C_VEL
LIN {X 0,Y 382.996,Z 636.901,A -85,B 0,C 180,E1 -12104.303,E2 -12104.303} C_VEL
LIN {X 0,Y 383.013,Z 636.906,A -85,B 0,C 180,E1 -12107.241,E2 -12107.241} C_VEL
LIN {X 0,Y 382.989,Z 636.905,A -85,B 0,C 180,E1 -12110.419,E2 -12110.419} C_VEL
LIN {X 0,Y 383.018,Z 636.896,A -85,B 0,C 180,E1 -12114.044,E2 -12114.044} C_VEL
LIN {X 0,Y 383.026,Z 636.965,A -85,B 0,C 180,E1 -12117.026,E2 -12117.026} C_VEL
LIN {X 0,Y 384.89,Z 644.905,A -85,B 0,C 180,E1 -12119.174,E2 -12119.174} C_VEL
LIN {X 0,Y 393.528,Z 664.806,A -85,B 0,C 180,E1 -12120.24,E2 -12120.24} C_VEL
LIN {X 0,Y 395.008,Z 669.605,A -85,B 0,C 180,E1 -12120.444,E2 -12120.444} C_VEL
LIN {X 0,Y 395.624,Z 672.888,A -85,B 0,C 180,E1 -12120.554,E2 -12120.554} C_VEL
LIN {X 0,Y 393.575,Z 780.074,A -85,B 0,C 180,E1 -12122.553,E2 -12122.553} C_VEL
LIN {X 0,Y 392.878,Z 794.515,A -85,B 0,C 180,E1 -12123.005,E2 -12123.005} C_VEL
LIN {X 0,Y 392.041,Z 807.682,A -85,B 0,C 180,E1 -12123.619,E2 -12123.619} C_VEL
LIN {X 0,Y 391.141,Z 818.934,A -85,B 0,C 180,E1 -12124.307,E2 -12124.307} C_VEL
LIN {X 0,Y 390.021,Z 830.93,A -85,B 0,C 180,E1 -12125.231,E2 -12125.231} C_VEL
LIN {X 0,Y 388.733,Z 843.279,A -85,B 0,C 180,E1 -12126.422,E2 -12126.422} C_VEL
LIN {X 0,Y 387.479,Z 853.878,A -85,B 0,C 180,E1 -12127.674,E2 -12127.674} C_VEL
LIN {X 0,Y 386.192,Z 864.545,A -85,B 0,C 180,E1 -12129.215,E2 -12129.215} C_VEL
LIN {X 0,Y 384.978,Z 873.68,A -85,B 0,C 180,E1 -12130.816,E2 -12130.816} C_VEL
LIN {X 0,Y 384.076,Z 881.465,A -85,B 0,C 180,E1 -12132.477,E2 -12132.477} C_VEL
LIN {X 0,Y 383.277,Z 887.559,A -85,B 0,C 180,E1 -12134.035,E2 -12134.035} C_VEL
LIN {X 0,Y 382.693,Z 892.709,A -85,B 0,C 180,E1 -12135.646,E2 -12135.646} C_VEL
LIN {X 0,Y 382.135,Z 898.101,A -85,B 0,C 180,E1 -12137.79,E2 -12137.79} C_VEL
LIN {X 0,Y 381.839,Z 901.071,A -85,B 0,C 180,E1 -12139.394,E2 -12139.394} C_VEL
LIN {X 0,Y 381.686,Z 903.812,A -85,B 0,C 180,E1 -12141.529,E2 -12141.529} C_VEL
LIN {X 0,Y 381.7,Z 905.187,A -85,B 0,C 180,E1 -12143.657,E2 -12143.657} C_VEL
LIN {X 0,Y 381.608,Z 905.249,A -85,B 0,C 180,E1 -12145.775,E2 -12145.775} C_VEL
LIN {X 0,Y 381.697,Z 903.987,A -85,B 0,C 180,E1 -12147.89,E2 -12147.89} C_VEL
LIN {X 0,Y 381.721,Z 901.388,A -85,B 0,C 180,E1 -12150,E2 -12150} C_VEL
LIN {X 0,Y 381.952,Z 897.378,A -85,B 0,C 180,E1 -12152.109,E2 -12152.109} C_VEL
LIN {X 0,Y 382.545,Z 891.829,A -85,B 0,C 180,E1 -12154.214,E2 -12154.214} C_VEL
LIN {X 0,Y 383.099,Z 886.571,A -85,B 0,C 180,E1 -12155.791,E2 -12155.791} C_VEL
LIN {X 0,Y 383.505,Z 882.312,A -85,B 0,C 180,E1 -12156.875,E2 -12156.875} C_VEL
LIN {X 0,Y 383.287,Z 879.188,A -85,B 0,C 180,E1 -12157.617,E2 -12157.617} C_VEL
LIN {X 0,Y 381.048,Z 873.87,A -85,B 0,C 180,E1 -12158.823,E2 -12158.823} C_VEL
LIN {X 0,Y 378.805,Z 868.16,A -85,B 0,C 180,E1 -12159.995,E2 -12159.995} C_VEL
LIN {X 0,Y 378.59,Z 864.228,A -85,B 0,C 180,E1 -12160.674,E2 -12160.674} C_VEL
LIN {X 0,Y 379.695,Z 854.996,A -85,B 0,C 180,E1 -12162.019,E2 -12162.019} C_VEL
LIN {X 0,Y 380.838,Z 844.167,A -85,B 0,C 180,E1 -12163.337,E2 -12163.337} C_VEL
LIN {X 0,Y 381.987,Z 832.303,A -85,B 0,C 180,E1 -12164.518,E2 -12164.518} C_VEL
LIN {X 0,Y 382.972,Z 820.921,A -85,B 0,C 180,E1 -12165.432,E2 -12165.432} C_VEL
LIN {X 0,Y 383.99,Z 807.592,A -85,B 0,C 180,E1 -12166.276,E2 -12166.276} C_VEL
LIN {X 0,Y 384.717,Z 793.729,A -85,B 0,C 180,E1 -12166.927,E2 -12166.927} C_VEL
LIN {X 0,Y 385.248,Z 780.488,A -85,B 0,C 180,E1 -12167.347,E2 -12167.347} C_VEL
LIN {X 0,Y 387.194,Z 672.604,A -85,B 0,C 180,E1 -12169.373,E2 -12169.373} C_VEL
LIN {X 0,Y 385.192,Z 664.491,A -85,B 0,C 180,E1 -12169.659,E2 -12169.659} C_VEL
LIN {X 0,Y 377.56,Z 644.873,A -85,B 0,C 180,E1 -12170.566,E2 -12170.566} C_VEL
LIN {X 0,Y 375.976,Z 637.78,A -85,B 0,C 180,E1 -12172.46,E2 -12172.46} C_VEL
LIN {X 0,Y 375.95,Z 637.78,A -85,B 0,C 180,E1 -12176.192,E2 -12176.192} C_VEL
LIN {X 0,Y 375.916,Z 637.783,A -85,B 0,C 180,E1 -12179.084,E2 -12179.084} C_VEL
LIN {X 0,Y 375.938,Z 637.781,A -85,B 0,C 180,E1 -12181.564,E2 -12181.564} C_VEL
LIN {X 0,Y 375.977,Z 637.777,A -85,B 0,C 180,E1 -12184.666,E2 -12184.666} C_VEL
LIN {X 0,Y 375.938,Z 637.78,A -85,B 0,C 180,E1 -12188.263,E2 -12188.263} C_VEL
LIN {X 0,Y 375.92,Z 637.782,A -85,B 0,C 180,E1 -12191.597,E2 -12191.597} C_VEL
LIN {X 0,Y 375.924,Z 637.78,A -85,B 0,C 180,E1 -12194.73,E2 -12194.73} C_VEL
LIN {X 0,Y 375.919,Z 637.781,A -85,B 0,C 180,E1 -12197.697,E2 -12197.697} C_VEL
LIN {X 0,Y 375.937,Z 637.778,A -85,B 0,C 180,E1 -12200.534,E2 -12200.534} C_VEL
LIN {X 0,Y 375.961,Z 637.76,A -85,B 0,C 180,E1 -12203.497,E2 -12203.497} C_VEL
LIN {X 0,Y 375.961,Z 637.776,A -85,B 0,C 180,E1 -12205.888,E2 -12205.888} C_VEL
LIN {X 0,Y 375.965,Z 637.768,A -85,B 0,C 180,E1 -12209.687,E2 -12209.687} C_VEL
LIN {X 0,Y 375.93,Z 637.78,A -85,B 0,C 180,E1 -12212.136,E2 -12212.136} C_VEL
LIN {X 0,Y 375.971,Z 637.766,A -85,B 0,C 180,E1 -12215.716,E2 -12215.716} C_VEL
LIN {X 0,Y 376.001,Z 637.774,A -85,B 0,C 180,E1 -12219.198,E2 -12219.198} C_VEL
LIN {X 0,Y 376.035,Z 637.752,A -85,B 0,C 180,E1 -12222.6,E2 -12222.6} C_VEL
LIN {X 0,Y 376.092,Z 637.759,A -85,B 0,C 180,E1 -12226.342,E2 -12226.342} C_VEL
LIN {X 0,Y 376.116,Z 637.749,A -85,B 0,C 180,E1 -12230.318,E2 -12230.318} C_VEL
LIN {X 0,Y 376.203,Z 637.751,A -85,B 0,C 180,E1 -12233.564,E2 -12233.564} C_VEL
LIN {X 0,Y 376.352,Z 637.732,A -85,B 0,C 180,E1 -12237.859,E2 -12237.859} C_VEL
LIN {X 0,Y 376.488,Z 637.708,A -85,B 0,C 180,E1 -12240,E2 -12240} C_VEL
LIN {X 0,Y 376.186,Z 637.748,A -85,B 0,C 180,E1 -12243.213,E2 -12243.213} C_VEL
LIN {X 0,Y 376.224,Z 637.742,A -85,B 0,C 180,E1 -12246.435,E2 -12246.435} C_VEL
LIN {X 0,Y 376.121,Z 637.759,A -85,B 0,C 180,E1 -12249.681,E2 -12249.681} C_VEL
LIN {X 0,Y 376.091,Z 637.762,A -85,B 0,C 180,E1 -12253.657,E2 -12253.657} C_VEL
LIN {X 0,Y 376.054,Z 637.763,A -85,B 0,C 180,E1 -12257.399,E2 -12257.399} C_VEL
LIN {X 0,Y 375.98,Z 637.772,A -85,B 0,C 180,E1 -12260.832,E2 -12260.832} C_VEL
LIN {X 0,Y 375.99,Z 637.772,A -85,B 0,C 180,E1 -12264.282,E2 -12264.282} C_VEL
LIN {X 0,Y 376.021,Z 637.766,A -85,B 0,C 180,E1 -12266.652,E2 -12266.652} C_VEL
LIN {X 0,Y 375.972,Z 637.774,A -85,B 0,C 180,E1 -12269.079,E2 -12269.079} C_VEL
LIN {X 0,Y 375.957,Z 637.777,A -85,B 0,C 180,E1 -12272.827,E2 -12272.827} C_VEL
LIN {X 0,Y 375.96,Z 637.777,A -85,B 0,C 180,E1 -12275.415,E2 -12275.415} C_VEL
LIN {X 0,Y 375.979,Z 637.778,A -85,B 0,C 180,E1 -12278.271,E2 -12278.271} C_VEL
LIN {X 0,Y 375.961,Z 637.775,A -85,B 0,C 180,E1 -12281.605,E2 -12281.605} C_VEL
LIN {X 0,Y 375.93,Z 637.779,A -85,B 0,C 180,E1 -12285.268,E2 -12285.268} C_VEL
LIN {X 0,Y 375.937,Z 637.782,A -85,B 0,C 180,E1 -12288.399,E2 -12288.399} C_VEL
LIN {X 0,Y 375.977,Z 637.776,A -85,B 0,C 180,E1 -12291.729,E2 -12291.729} C_VEL
LIN {X 0,Y 375.981,Z 637.778,A -85,B 0,C 180,E1 -12295.332,E2 -12295.332} C_VEL
LIN {X 0,Y 375.966,Z 637.934,A -85,B 0,C 180,E1 -12297.61,E2 -12297.61} C_VEL
LIN {X 0,Y 379.282,Z 652.015,A -85,B 0,C 180,E1 -12300.817,E2 -12300.817} C_VEL
LIN {X 0,Y 381.231,Z 661.334,A -85,B 0,C 180,E1 -12302.853,E2 -12302.853} C_VEL
LIN {X 0,Y 381.089,Z 665.724,A -85,B 0,C 180,E1 -12303.73,E2 -12303.73} C_VEL
LIN {X 0,Y 380.668,Z 670.486,A -85,B 0,C 180,E1 -12304.659,E2 -12304.659} C_VEL
LIN {X 0,Y 386.754,Z 706.442,A -85,B 0,C 180,E1 -12305.762,E2 -12305.762} C_VEL
LIN {X 0,Y 385.012,Z 806.484,A -85,B 0,C 180,E1 -12307.636,E2 -12307.636} C_VEL
LIN {X 0,Y 384.385,Z 820.543,A -85,B 0,C 180,E1 -12308.057,E2 -12308.057} C_VEL
LIN {X 0,Y 383.43,Z 834.919,A -85,B 0,C 180,E1 -12308.706,E2 -12308.706} C_VEL
LIN {X 0,Y 382.364,Z 848.552,A -85,B 0,C 180,E1 -12309.56,E2 -12309.56} C_VEL
LIN {X 0,Y 381.146,Z 861.602,A -85,B 0,C 180,E1 -12310.615,E2 -12310.615} C_VEL
LIN {X 0,Y 379.855,Z 873.434,A -85,B 0,C 180,E1 -12311.807,E2 -12311.807} C_VEL
LIN {X 0,Y 378.778,Z 883.275,A -85,B 0,C 180,E1 -12313.008,E2 -12313.008} C_VEL
LIN {X 0,Y 377.525,Z 894.154,A -85,B 0,C 180,E1 -12314.616,E2 -12314.616} C_VEL
LIN {X 0,Y 376.616,Z 902.878,A -85,B 0,C 180,E1 -12316.183,E2 -12316.183} C_VEL
LIN {X 0,Y 375.91,Z 910.614,A -85,B 0,C 180,E1 -12317.858,E2 -12317.858} C_VEL
LIN {X 0,Y 375.191,Z 917.752,A -85,B 0,C 180,E1 -12319.749,E2 -12319.749} C_VEL
LIN {X 0,Y 374.79,Z 924.165,A -85,B 0,C 180,E1 -12321.915,E2 -12321.915} C_VEL
LIN {X 0,Y 374.661,Z 928.411,A -85,B 0,C 180,E1 -12323.82,E2 -12323.82} C_VEL
LIN {X 0,Y 374.544,Z 931.445,A -85,B 0,C 180,E1 -12325.695,E2 -12325.695} C_VEL
LIN {X 0,Y 374.512,Z 933.628,A -85,B 0,C 180,E1 -12327.849,E2 -12327.849} C_VEL
LIN {X 0,Y 374.587,Z 934.454,A -85,B 0,C 180,E1 -12330,E2 -12330} C_VEL
LIN {X 0,Y 374.493,Z 933.932,A -85,B 0,C 180,E1 -12332.151,E2 -12332.151} C_VEL
LIN {X 0,Y 374.543,Z 932.074,A -85,B 0,C 180,E1 -12334.304,E2 -12334.304} C_VEL
LIN {X 0,Y 374.628,Z 928.827,A -85,B 0,C 180,E1 -12336.463,E2 -12336.463} C_VEL
LIN {X 0,Y 374.873,Z 924.076,A -85,B 0,C 180,E1 -12338.626,E2 -12338.626} C_VEL
LIN {X 0,Y 375.379,Z 917.702,A -85,B 0,C 180,E1 -12340.791,E2 -12340.791} C_VEL
LIN {X 0,Y 376.246,Z 910.631,A -85,B 0,C 180,E1 -12342.678,E2 -12342.678} C_VEL
LIN {X 0,Y 377.216,Z 902.163,A -85,B 0,C 180,E1 -12344.512,E2 -12344.512} C_VEL
LIN {X 0,Y 378.331,Z 892.772,A -85,B 0,C 180,E1 -12346.179,E2 -12346.179} C_VEL
LIN {X 0,Y 379.771,Z 881.752,A -85,B 0,C 180,E1 -12347.779,E2 -12347.779} C_VEL
LIN {X 0,Y 381.248,Z 870.544,A -85,B 0,C 180,E1 -12349.099,E2 -12349.099} C_VEL
LIN {X 0,Y 382.655,Z 858.177,A -85,B 0,C 180,E1 -12350.283,E2 -12350.283} C_VEL
LIN {X 0,Y 383.916,Z 845.471,A -85,B 0,C 180,E1 -12351.253,E2 -12351.253} C_VEL
LIN {X 0,Y 385.103,Z 832.038,A -85,B 0,C 180,E1 -12352.04,E2 -12352.04} C_VEL
LIN {X 0,Y 386.097,Z 818.532,A -85,B 0,C 180,E1 -12352.615,E2 -12352.615} C_VEL
LIN {X 0,Y 386.701,Z 803.541,A -85,B 0,C 180,E1 -12353.036,E2 -12353.036} C_VEL
LIN {X 0,Y 388.663,Z 707.194,A -85,B 0,C 180,E1 -12354.843,E2 -12354.843} C_VEL
LIN {X 0,Y 384.217,Z 682.674,A -85,B 0,C 180,E1 -12355.677,E2 -12355.677} C_VEL
LIN {X 0,Y 381.685,Z 670.113,A -85,B 0,C 180,E1 -12356.166,E2 -12356.166} C_VEL
LIN {X 0,Y 382.203,Z 665.573,A -85,B 0,C 180,E1 -12357.072,E2 -12357.072} C_VEL
LIN {X 0,Y 381.194,Z 659.547,A -85,B 0,C 180,E1 -12358.414,E2 -12358.414} C_VEL
LIN {X 0,Y 379.033,Z 649.9,A -85,B 0,C 180,E1 -12360.657,E2 -12360.657} C_VEL
LIN {X 0,Y 375.966,Z 637.77,A -85,B 0,C 180,E1 -12363.667,E2 -12363.667} C_VEL
LIN {X 0,Y 375.955,Z 637.777,A -85,B 0,C 180,E1 -12366.741,E2 -12366.741} C_VEL
LIN {X 0,Y 375.997,Z 637.768,A -85,B 0,C 180,E1 -12369.972,E2 -12369.972} C_VEL
LIN {X 0,Y 375.94,Z 637.772,A -85,B 0,C 180,E1 -12373.764,E2 -12373.764} C_VEL
LIN {X 0,Y 375.961,Z 637.767,A -85,B 0,C 180,E1 -12377.704,E2 -12377.704} C_VEL
LIN {X 0,Y 375.969,Z 637.776,A -85,B 0,C 180,E1 -12380.538,E2 -12380.538} C_VEL
LIN {X 0,Y 375.966,Z 637.764,A -85,B 0,C 180,E1 -12383.495,E2 -12383.495} C_VEL
LIN {X 0,Y 375.962,Z 637.777,A -85,B 0,C 180,E1 -12385.889,E2 -12385.889} C_VEL
LIN {X 0,Y 375.965,Z 637.76,A -85,B 0,C 180,E1 -12389.688,E2 -12389.688} C_VEL
LIN {X 0,Y 375.996,Z 637.772,A -85,B 0,C 180,E1 -12392.142,E2 -12392.142} C_VEL
LIN {X 0,Y 376.007,Z 637.769,A -85,B 0,C 180,E1 -12394.539,E2 -12394.539} C_VEL
LIN {X 0,Y 375.964,Z 637.773,A -85,B 0,C 180,E1 -12398.046,E2 -12398.046} C_VEL
LIN {X 0,Y 376.025,Z 637.766,A -85,B 0,C 180,E1 -12401.474,E2 -12401.474} C_VEL
LIN {X 0,Y 376.062,Z 637.762,A -85,B 0,C 180,E1 -12404.833,E2 -12404.833} C_VEL
LIN {X 0,Y 376.052,Z 637.769,A -85,B 0,C 180,E1 -12408.137,E2 -12408.137} C_VEL
LIN {X 0,Y 376.22,Z 637.74,A -85,B 0,C 180,E1 -12411.919,E2 -12411.919} C_VEL
LIN {X 0,Y 376.171,Z 637.746,A -85,B 0,C 180,E1 -12414.64,E2 -12414.64} C_VEL
LIN {X 0,Y 376.353,Z 637.728,A -85,B 0,C 180,E1 -12417.86,E2 -12417.86} C_VEL
LIN {X 0,Y 376.489,Z 637.709,A -85,B 0,C 180,E1 -12420,E2 -12420} C_VEL
LIN {X 0,Y 376.187,Z 637.748,A -85,B 0,C 180,E1 -12423.213,E2 -12423.213} C_VEL
LIN {X 0,Y 376.23,Z 637.739,A -85,B 0,C 180,E1 -12426.553,E2 -12426.553} C_VEL
LIN {X 0,Y 376.121,Z 637.753,A -85,B 0,C 180,E1 -12429.682,E2 -12429.682} C_VEL
LIN {X 0,Y 376.091,Z 637.759,A -85,B 0,C 180,E1 -12433.658,E2 -12433.658} C_VEL
LIN {X 0,Y 376.046,Z 637.766,A -85,B 0,C 180,E1 -12437.608,E2 -12437.608} C_VEL
LIN {X 0,Y 375.98,Z 637.777,A -85,B 0,C 180,E1 -12440.832,E2 -12440.832} C_VEL
LIN {X 0,Y 375.981,Z 637.77,A -85,B 0,C 180,E1 -12444.283,E2 -12444.283} C_VEL
LIN {X 0,Y 375.944,Z 637.778,A -85,B 0,C 180,E1 -12446.658,E2 -12446.658} C_VEL
LIN {X 0,Y 375.964,Z 637.763,A -85,B 0,C 180,E1 -12450.313,E2 -12450.313} C_VEL
LIN {X 0,Y 375.962,Z 637.772,A -85,B 0,C 180,E1 -12454.112,E2 -12454.112} C_VEL
LIN {X 0,Y 375.954,Z 637.778,A -85,B 0,C 180,E1 -12456.742,E2 -12456.742} C_VEL
LIN {X 0,Y 375.941,Z 637.772,A -85,B 0,C 180,E1 -12459.962,E2 -12459.962} C_VEL
LIN {X 0,Y 375.931,Z 637.782,A -85,B 0,C 180,E1 -12463.767,E2 -12463.767} C_VEL
LIN {X 0,Y 375.934,Z 637.783,A -85,B 0,C 180,E1 -12466.811,E2 -12466.811} C_VEL
LIN {X 0,Y 375.938,Z 637.784,A -85,B 0,C 180,E1 -12470.534,E2 -12470.534} C_VEL
LIN {X 0,Y 375.961,Z 637.779,A -85,B 0,C 180,E1 -12473.497,E2 -12473.497} C_VEL
LIN {X 0,Y 376.011,Z 637.909,A -85,B 0,C 180,E1 -12476.579,E2 -12476.579} C_VEL
LIN {X 0,Y 377.768,Z 645.274,A -85,B 0,C 180,E1 -12478.607,E2 -12478.607} C_VEL
LIN {X 0,Y 385.977,Z 663.796,A -85,B 0,C 180,E1 -12479.649,E2 -12479.649} C_VEL
LIN {X 0,Y 388.612,Z 670.663,A -85,B 0,C 180,E1 -12479.991,E2 -12479.991} C_VEL
LIN {X 0,Y 389.255,Z 674.311,A -85,B 0,C 180,E1 -12480.114,E2 -12480.114} C_VEL
LIN {X 0,Y 387.131,Z 780.664,A -85,B 0,C 180,E1 -12482.13,E2 -12482.13} C_VEL
LIN {X 0,Y 386.399,Z 794.948,A -85,B 0,C 180,E1 -12482.587,E2 -12482.587} C_VEL
LIN {X 0,Y 385.433,Z 809.005,A -85,B 0,C 180,E1 -12483.264,E2 -12483.264} C_VEL
LIN {X 0,Y 384.49,Z 820.315,A -85,B 0,C 180,E1 -12483.98,E2 -12483.98} C_VEL
LIN {X 0,Y 383.155,Z 833.493,A -85,B 0,C 180,E1 -12485.047,E2 -12485.047} C_VEL
LIN {X 0,Y 381.825,Z 845.383,A -85,B 0,C 180,E1 -12486.257,E2 -12486.257} C_VEL
LIN {X 0,Y 380.422,Z 857.095,A -85,B 0,C 180,E1 -12487.73,E2 -12487.73} C_VEL
LIN {X 0,Y 379.014,Z 867.719,A -85,B 0,C 180,E1 -12489.371,E2 -12489.371} C_VEL
LIN {X 0,Y 377.821,Z 876.363,A -85,B 0,C 180,E1 -12491.003,E2 -12491.003} C_VEL
LIN {X 0,Y 376.785,Z 884.6,A -85,B 0,C 180,E1 -12492.916,E2 -12492.916} C_VEL
LIN {X 0,Y 375.893,Z 891.189,A -85,B 0,C 180,E1 -12494.826,E2 -12494.826} C_VEL
LIN {X 0,Y 375.237,Z 897.009,A -85,B 0,C 180,E1 -12497.012,E2 -12497.012} C_VEL
LIN {X 0,Y 374.798,Z 901.243,A -85,B 0,C 180,E1 -12499.192,E2 -12499.192} C_VEL
LIN {X 0,Y 374.618,Z 904.021,A -85,B 0,C 180,E1 -12501.368,E2 -12501.368} C_VEL
LIN {X 0,Y 374.616,Z 905.433,A -85,B 0,C 180,E1 -12503.537,E2 -12503.537} C_VEL
LIN {X 0,Y 374.535,Z 905.531,A -85,B 0,C 180,E1 -12505.696,E2 -12505.696} C_VEL
LIN {X 0,Y 374.595,Z 904.314,A -85,B 0,C 180,E1 -12507.85,E2 -12507.85} C_VEL
LIN {X 0,Y 374.65,Z 901.761,A -85,B 0,C 180,E1 -12510,E2 -12510} C_VEL
LIN {X 0,Y 374.888,Z 897.792,A -85,B 0,C 180,E1 -12512.149,E2 -12512.149} C_VEL
LIN {X 0,Y 375.501,Z 892.284,A -85,B 0,C 180,E1 -12514.294,E2 -12514.294} C_VEL
LIN {X 0,Y 376.068,Z 887.073,A -85,B 0,C 180,E1 -12515.9,E2 -12515.9} C_VEL
LIN {X 0,Y 376.953,Z 879.571,A -85,B 0,C 180,E1 -12517.769,E2 -12517.769} C_VEL
LIN {X 0,Y 377.597,Z 872.053,A -85,B 0,C 180,E1 -12519.324,E2 -12519.324} C_VEL
LIN {X 0,Y 378.59,Z 864.228,A -85,B 0,C 180,E1 -12520.674,E2 -12520.674} C_VEL
LIN {X 0,Y 378.424,Z 860.226,A -85,B 0,C 180,E1 -12521.334,E2 -12521.334} C_VEL
LIN {X 0,Y 376.419,Z 853.516,A -85,B 0,C 180,E1 -12522.405,E2 -12522.405} C_VEL
LIN {X 0,Y 374.463,Z 846.347,A -85,B 0,C 180,E1 -12523.408,E2 -12523.408} C_VEL
LIN {X 0,Y 374.362,Z 841.628,A -85,B 0,C 180,E1 -12523.951,E2 -12523.951} C_VEL
LIN {X 0,Y 375.452,Z 830.218,A -85,B 0,C 180,E1 -12525.054,E2 -12525.054} C_VEL
LIN {X 0,Y 376.519,Z 818.297,A -85,B 0,C 180,E1 -12525.981,E2 -12525.981} C_VEL
LIN {X 0,Y 377.475,Z 805.228,A -85,B 0,C 180,E1 -12526.773,E2 -12526.773} C_VEL
LIN {X 0,Y 378.215,Z 791.084,A -85,B 0,C 180,E1 -12527.401,E2 -12527.401} C_VEL
LIN {X 0,Y 378.653,Z 777.489,A -85,B 0,C 180,E1 -12527.799,E2 -12527.799} C_VEL
LIN {X 0,Y 380.638,Z 673.835,A -85,B 0,C 180,E1 -12529.764,E2 -12529.764} C_VEL
LIN {X 0,Y 379.065,Z 667.277,A -85,B 0,C 180,E1 -12529.998,E2 -12529.998} C_VEL
LIN {X 0,Y 371.271,Z 647.518,A -85,B 0,C 180,E1 -12530.93,E2 -12530.93} C_VEL
LIN {X 0,Y 370.35,Z 645.041,A -85,B 0,C 180,E1 -12531.083,E2 -12531.083} C_VEL
LIN {X 0,Y 368.934,Z 638.657,A -85,B 0,C 180,E1 -12532.839,E2 -12532.839} C_VEL
LIN {X 0,Y 368.882,Z 638.66,A -85,B 0,C 180,E1 -12536.432,E2 -12536.432} C_VEL
LIN {X 0,Y 368.895,Z 638.659,A -85,B 0,C 180,E1 -12539.692,E2 -12539.692} C_VEL
LIN {X 0,Y 368.897,Z 638.658,A -85,B 0,C 180,E1 -12543.538,E2 -12543.538} C_VEL
LIN {X 0,Y 368.898,Z 638.659,A -85,B 0,C 180,E1 -12546.854,E2 -12546.854} C_VEL
LIN {X 0,Y 368.886,Z 638.645,A -85,B 0,C 180,E1 -12550.374,E2 -12550.374} C_VEL
LIN {X 0,Y 368.881,Z 638.655,A -85,B 0,C 180,E1 -12553.615,E2 -12553.615} C_VEL
LIN {X 0,Y 368.886,Z 638.66,A -85,B 0,C 180,E1 -12556.695,E2 -12556.695} C_VEL
LIN {X 0,Y 368.887,Z 638.657,A -85,B 0,C 180,E1 -12559.648,E2 -12559.648} C_VEL
LIN {X 0,Y 368.899,Z 638.636,A -85,B 0,C 180,E1 -12563.145,E2 -12563.145} C_VEL
LIN {X 0,Y 368.899,Z 638.655,A -85,B 0,C 180,E1 -12566.462,E2 -12566.462} C_VEL
LIN {X 0,Y 368.932,Z 638.648,A -85,B 0,C 180,E1 -12569.046,E2 -12569.046} C_VEL
LIN {X 0,Y 368.869,Z 638.66,A -85,B 0,C 180,E1 -12572.789,E2 -12572.789} C_VEL
LIN {X 0,Y 368.948,Z 638.639,A -85,B 0,C 180,E1 -12576.42,E2 -12576.42} C_VEL
LIN {X 0,Y 368.939,Z 638.65,A -85,B 0,C 180,E1 -12579.947,E2 -12579.947} C_VEL
LIN {X 0,Y 368.971,Z 638.637,A -85,B 0,C 180,E1 -12583.398,E2 -12583.398} C_VEL
LIN {X 0,Y 369.061,Z 638.635,A -85,B 0,C 180,E1 -12586.79,E2 -12586.79} C_VEL
LIN {X 0,Y 369.066,Z 638.626,A -85,B 0,C 180,E1 -12590.131,E2 -12590.131} C_VEL
LIN {X 0,Y 369.164,Z 638.626,A -85,B 0,C 180,E1 -12593.441,E2 -12593.441} C_VEL
LIN {X 0,Y 369.317,Z 638.608,A -85,B 0,C 180,E1 -12597.819,E2 -12597.819} C_VEL
LIN {X 0,Y 369.457,Z 638.584,A -85,B 0,C 180,E1 -12600,E2 -12600} C_VEL
LIN {X 0,Y 369.318,Z 638.606,A -85,B 0,C 180,E1 -12602.181,E2 -12602.181} C_VEL
LIN {X 0,Y 369.185,Z 638.618,A -85,B 0,C 180,E1 -12606.558,E2 -12606.558} C_VEL
LIN {X 0,Y 369.109,Z 638.629,A -85,B 0,C 180,E1 -12608.761,E2 -12608.761} C_VEL
LIN {X 0,Y 369.008,Z 638.644,A -85,B 0,C 180,E1 -12612.093,E2 -12612.093} C_VEL
LIN {X 0,Y 369.003,Z 638.638,A -85,B 0,C 180,E1 -12615.464,E2 -12615.464} C_VEL
LIN {X 0,Y 368.985,Z 638.64,A -85,B 0,C 180,E1 -12618.892,E2 -12618.892} C_VEL
LIN {X 0,Y 368.924,Z 638.652,A -85,B 0,C 180,E1 -12622.395,E2 -12622.395} C_VEL
LIN {X 0,Y 369.001,Z 638.645,A -85,B 0,C 180,E1 -12625.98,E2 -12625.98} C_VEL
LIN {X 0,Y 368.963,Z 638.649,A -85,B 0,C 180,E1 -12628.811,E2 -12628.811} C_VEL
LIN {X 0,Y 368.904,Z 638.659,A -85,B 0,C 180,E1 -12632.237,E2 -12632.237} C_VEL
LIN {X 0,Y 368.931,Z 638.653,A -85,B 0,C 180,E1 -12635.001,E2 -12635.001} C_VEL
LIN {X 0,Y 368.914,Z 638.656,A -85,B 0,C 180,E1 -12638.641,E2 -12638.641} C_VEL
LIN {X 0,Y 368.911,Z 638.654,A -85,B 0,C 180,E1 -12641.818,E2 -12641.818} C_VEL
LIN {X 0,Y 368.887,Z 638.657,A -85,B 0,C 180,E1 -12645.177,E2 -12645.177} C_VEL
LIN {X 0,Y 368.885,Z 638.658,A -85,B 0,C 180,E1 -12648.178,E2 -12648.178} C_VEL
LIN {X 0,Y 368.912,Z 638.656,A -85,B 0,C 180,E1 -12651.359,E2 -12651.359} C_VEL
LIN {X 0,Y 368.938,Z 638.655,A -85,B 0,C 180,E1 -12655.146,E2 -12655.146} C_VEL
LIN {X 0,Y 368.928,Z 638.818,A -85,B 0,C 180,E1 -12657.217,E2 -12657.217} C_VEL
LIN {X 0,Y 372.091,Z 652.113,A -85,B 0,C 180,E1 -12660.324,E2 -12660.324} C_VEL
LIN {X 0,Y 374.24,Z 662.38,A -85,B 0,C 180,E1 -12662.619,E2 -12662.619} C_VEL
LIN {X 0,Y 374.33,Z 665.254,A -85,B 0,C 180,E1 -12663.218,E2 -12663.218} C_VEL
LIN {X 0,Y 373.87,Z 670.197,A -85,B 0,C 180,E1 -12664.204,E2 -12664.204} C_VEL
LIN {X 0,Y 380.196,Z 707.523,A -85,B 0,C 180,E1 -12665.38,E2 -12665.38} C_VEL
LIN {X 0,Y 378.454,Z 803.175,A -85,B 0,C 180,E1 -12667.191,E2 -12667.191} C_VEL
LIN {X 0,Y 377.836,Z 817.498,A -85,B 0,C 180,E1 -12667.585,E2 -12667.585} C_VEL
LIN {X 0,Y 376.941,Z 831.399,A -85,B 0,C 180,E1 -12668.177,E2 -12668.177} C_VEL
LIN {X 0,Y 375.903,Z 844.917,A -85,B 0,C 180,E1 -12668.977,E2 -12668.977} C_VEL
LIN {X 0,Y 374.657,Z 857.975,A -85,B 0,C 180,E1 -12669.981,E2 -12669.981} C_VEL
LIN {X 0,Y 373.392,Z 870.477,A -85,B 0,C 180,E1 -12671.196,E2 -12671.196} C_VEL
LIN {X 0,Y 372.037,Z 881.771,A -85,B 0,C 180,E1 -12672.549,E2 -12672.549} C_VEL
LIN {X 0,Y 370.825,Z 892.033,A -85,B 0,C 180,E1 -12674.049,E2 -12674.049} C_VEL
LIN {X 0,Y 369.751,Z 901.325,A -85,B 0,C 180,E1 -12675.694,E2 -12675.694} C_VEL
LIN {X 0,Y 368.994,Z 909.071,A -85,B 0,C 180,E1 -12677.348,E2 -12677.348} C_VEL
LIN {X 0,Y 368.317,Z 915.509,A -85,B 0,C 180,E1 -12679,E2 -12679} C_VEL
LIN {X 0,Y 367.896,Z 920.804,A -85,B 0,C 180,E1 -12680.655,E2 -12680.655} C_VEL
LIN {X 0,Y 367.577,Z 926.391,A -85,B 0,C 180,E1 -12682.861,E2 -12682.861} C_VEL
LIN {X 0,Y 367.48,Z 929.5,A -85,B 0,C 180,E1 -12684.513,E2 -12684.513} C_VEL
LIN {X 0,Y 367.383,Z 932.4,A -85,B 0,C 180,E1 -12686.71,E2 -12686.71} C_VEL
LIN {X 0,Y 367.483,Z 933.923,A -85,B 0,C 180,E1 -12688.904,E2 -12688.904} C_VEL
LIN {X 0,Y 367.481,Z 934.093,A -85,B 0,C 180,E1 -12691.096,E2 -12691.096} C_VEL
LIN {X 0,Y 367.374,Z 932.921,A -85,B 0,C 180,E1 -12693.29,E2 -12693.29} C_VEL
LIN {X 0,Y 367.47,Z 930.4,A -85,B 0,C 180,E1 -12695.487,E2 -12695.487} C_VEL
LIN {X 0,Y 367.661,Z 926.446,A -85,B 0,C 180,E1 -12697.69,E2 -12697.69} C_VEL
LIN {X 0,Y 368.073,Z 920.925,A -85,B 0,C 180,E1 -12699.895,E2 -12699.895} C_VEL
LIN {X 0,Y 368.754,Z 914.712,A -85,B 0,C 180,E1 -12701.822,E2 -12701.822} C_VEL
LIN {X 0,Y 369.728,Z 906.982,A -85,B 0,C 180,E1 -12703.745,E2 -12703.745} C_VEL
LIN {X 0,Y 370.858,Z 897.448,A -85,B 0,C 180,E1 -12705.667,E2 -12705.667} C_VEL
LIN {X 0,Y 372.211,Z 887.479,A -85,B 0,C 180,E1 -12707.301,E2 -12707.301} C_VEL
LIN {X 0,Y 373.754,Z 876.415,A -85,B 0,C 180,E1 -12708.785,E2 -12708.785} C_VEL
LIN {X 0,Y 375.203,Z 865.434,A -85,B 0,C 180,E1 -12709.989,E2 -12709.989} C_VEL
LIN {X 0,Y 376.622,Z 853.158,A -85,B 0,C 180,E1 -12711.088,E2 -12711.088} C_VEL
LIN {X 0,Y 377.843,Z 840.545,A -85,B 0,C 180,E1 -12711.983,E2 -12711.983} C_VEL
LIN {X 0,Y 379.06,Z 826.367,A -85,B 0,C 180,E1 -12712.734,E2 -12712.734} C_VEL
LIN {X 0,Y 379.945,Z 812.349,A -85,B 0,C 180,E1 -12713.254,E2 -12713.254} C_VEL
LIN {X 0,Y 380.519,Z 794.741,A -85,B 0,C 180,E1 -12713.649,E2 -12713.649} C_VEL
LIN {X 0,Y 382.304,Z 708.01,A -85,B 0,C 180,E1 -12715.3,E2 -12715.3} C_VEL
LIN {X 0,Y 377.723,Z 682.876,A -85,B 0,C 180,E1 -12716.181,E2 -12716.181} C_VEL
LIN {X 0,Y 375.071,Z 669.918,A -85,B 0,C 180,E1 -12716.688,E2 -12716.688} C_VEL
LIN {X 0,Y 375.382,Z 666.91,A -85,B 0,C 180,E1 -12717.303,E2 -12717.303} C_VEL
LIN {X 0,Y 374.063,Z 659.786,A -85,B 0,C 180,E1 -12718.937,E2 -12718.937} C_VEL
LIN {X 0,Y 371.452,Z 648.573,A -85,B 0,C 180,E1 -12721.634,E2 -12721.634} C_VEL
LIN {X 0,Y 368.942,Z 638.648,A -85,B 0,C 180,E1 -12724.191,E2 -12724.191} C_VEL
LIN {X 0,Y 368.922,Z 638.655,A -85,B 0,C 180,E1 -12727.561,E2 -12727.561} C_VEL
LIN {X 0,Y 368.953,Z 638.644,A -85,B 0,C 180,E1 -12730.365,E2 -12730.365} C_VEL
LIN {X 0,Y 368.895,Z 638.65,A -85,B 0,C 180,E1 -12733.618,E2 -12733.618} C_VEL
LIN {X 0,Y 368.903,Z 638.655,A -85,B 0,C 180,E1 -12736.699,E2 -12736.699} C_VEL
LIN {X 0,Y 368.953,Z 638.651,A -85,B 0,C 180,E1 -12739.636,E2 -12739.636} C_VEL
LIN {X 0,Y 368.904,Z 638.64,A -85,B 0,C 180,E1 -12743.144,E2 -12743.144} C_VEL
LIN {X 0,Y 368.898,Z 638.653,A -85,B 0,C 180,E1 -12746.462,E2 -12746.462} C_VEL
LIN {X 0,Y 368.929,Z 638.63,A -85,B 0,C 180,E1 -12749.047,E2 -12749.047} C_VEL
LIN {X 0,Y 368.98,Z 638.646,A -85,B 0,C 180,E1 -12751.564,E2 -12751.564} C_VEL
LIN {X 0,Y 369,Z 638.64,A -85,B 0,C 180,E1 -12754.02,E2 -12754.02} C_VEL
LIN {X 0,Y 368.933,Z 638.647,A -85,B 0,C 180,E1 -12757.605,E2 -12757.605} C_VEL
LIN {X 0,Y 368.984,Z 638.642,A -85,B 0,C 180,E1 -12761.108,E2 -12761.108} C_VEL
LIN {X 0,Y 369.002,Z 638.643,A -85,B 0,C 180,E1 -12764.536,E2 -12764.536} C_VEL
LIN {X 0,Y 369.007,Z 638.643,A -85,B 0,C 180,E1 -12767.907,E2 -12767.907} C_VEL
LIN {X 0,Y 369.167,Z 638.618,A -85,B 0,C 180,E1 -12771.869,E2 -12771.869} C_VEL
LIN {X 0,Y 369.144,Z 638.623,A -85,B 0,C 180,E1 -12774.538,E2 -12774.538} C_VEL
LIN {X 0,Y 369.318,Z 638.604,A -85,B 0,C 180,E1 -12777.819,E2 -12777.819} C_VEL
LIN {X 0,Y 369.458,Z 638.584,A -85,B 0,C 180,E1 -12780,E2 -12780} C_VEL
LIN {X 0,Y 369.318,Z 638.603,A -85,B 0,C 180,E1 -12782.181,E2 -12782.181} C_VEL
LIN {X 0,Y 369.2,Z 638.616,A -85,B 0,C 180,E1 -12786.559,E2 -12786.559} C_VEL
LIN {X 0,Y 369.069,Z 638.632,A -85,B 0,C 180,E1 -12789.869,E2 -12789.869} C_VEL
LIN {X 0,Y 369.039,Z 638.638,A -85,B 0,C 180,E1 -12793.773,E2 -12793.773} C_VEL
LIN {X 0,Y 369.003,Z 638.643,A -85,B 0,C 180,E1 -12797.769,E2 -12797.769} C_VEL
LIN {X 0,Y 368.911,Z 638.656,A -85,B 0,C 180,E1 -12801.221,E2 -12801.221} C_VEL
LIN {X 0,Y 368.938,Z 638.652,A -85,B 0,C 180,E1 -12804.777,E2 -12804.777} C_VEL
LIN {X 0,Y 368.918,Z 638.636,A -85,B 0,C 180,E1 -12808.442,E2 -12808.442} C_VEL
LIN {X 0,Y 368.912,Z 638.648,A -85,B 0,C 180,E1 -12810.988,E2 -12810.988} C_VEL
LIN {X 0,Y 368.938,Z 638.651,A -85,B 0,C 180,E1 -12814.854,E2 -12814.854} C_VEL
LIN {X 0,Y 368.88,Z 638.662,A -85,B 0,C 180,E1 -12818.635,E2 -12818.635} C_VEL
LIN {X 0,Y 368.873,Z 638.657,A -85,B 0,C 180,E1 -12822.008,E2 -12822.008} C_VEL
LIN {X 0,Y 368.877,Z 638.654,A -85,B 0,C 180,E1 -12825.175,E2 -12825.175} C_VEL
LIN {X 0,Y 368.871,Z 638.663,A -85,B 0,C 180,E1 -12828.176,E2 -12828.176} C_VEL
LIN {X 0,Y 368.88,Z 638.664,A -85,B 0,C 180,E1 -12831.366,E2 -12831.366} C_VEL
LIN {X 0,Y 368.934,Z 638.654,A -85,B 0,C 180,E1 -12835.146,E2 -12835.146} C_VEL
LIN {X 0,Y 368.922,Z 638.662,A -85,B 0,C 180,E1 -12836.054,E2 -12836.054} C_VEL
LIN {X 0,Y 370.556,Z 645.53,A -85,B 0,C 180,E1 -12838.003,E2 -12838.003} C_VEL
LIN {X 0,Y 379.37,Z 665.009,A -85,B 0,C 180,E1 -12839.154,E2 -12839.154} C_VEL
LIN {X 0,Y 382.558,Z 673.109,A -85,B 0,C 180,E1 -12839.576,E2 -12839.576} C_VEL
LIN {X 0,Y 382.924,Z 675.982,A -85,B 0,C 180,E1 -12839.664,E2 -12839.664} C_VEL
LIN {X 0,Y 380.746,Z 779.764,A -85,B 0,C 180,E1 -12841.658,E2 -12841.658} C_VEL
LIN {X 0,Y 379.986,Z 794.602,A -85,B 0,C 180,E1 -12842.122,E2 -12842.122} C_VEL
LIN {X 0,Y 379.144,Z 807.356,A -85,B 0,C 180,E1 -12842.726,E2 -12842.726} C_VEL
LIN {X 0,Y 378.146,Z 818.361,A -85,B 0,C 180,E1 -12843.406,E2 -12843.406} C_VEL
LIN {X 0,Y 376.824,Z 831.641,A -85,B 0,C 180,E1 -12844.45,E2 -12844.45} C_VEL
LIN {X 0,Y 375.395,Z 843.947,A -85,B 0,C 180,E1 -12845.677,E2 -12845.677} C_VEL
LIN {X 0,Y 374.001,Z 855.01,A -85,B 0,C 180,E1 -12847.041,E2 -12847.041} C_VEL
LIN {X 0,Y 372.727,Z 864.355,A -85,B 0,C 180,E1 -12848.427,E2 -12848.427} C_VEL
LIN {X 0,Y 371.373,Z 873.613,A -85,B 0,C 180,E1 -12850.084,E2 -12850.084} C_VEL
LIN {X 0,Y 370.326,Z 881.338,A -85,B 0,C 180,E1 -12851.761,E2 -12851.761} C_VEL
LIN {X 0,Y 369.44,Z 887.671,A -85,B 0,C 180,E1 -12853.42,E2 -12853.42} C_VEL
LIN {X 0,Y 368.738,Z 892.891,A -85,B 0,C 180,E1 -12855.09,E2 -12855.09} C_VEL
LIN {X 0,Y 368.239,Z 897.143,A -85,B 0,C 180,E1 -12856.76,E2 -12856.76} C_VEL
LIN {X 0,Y 367.763,Z 901.416,A -85,B 0,C 180,E1 -12858.983,E2 -12858.983} C_VEL
LIN {X 0,Y 367.532,Z 904.232,A -85,B 0,C 180,E1 -12861.201,E2 -12861.201} C_VEL
LIN {X 0,Y 367.541,Z 905.68,A -85,B 0,C 180,E1 -12863.412,E2 -12863.412} C_VEL
LIN {X 0,Y 367.463,Z 905.812,A -85,B 0,C 180,E1 -12865.613,E2 -12865.613} C_VEL
LIN {X 0,Y 367.493,Z 904.634,A -85,B 0,C 180,E1 -12867.808,E2 -12867.808} C_VEL
LIN {X 0,Y 367.582,Z 902.127,A -85,B 0,C 180,E1 -12870,E2 -12870} C_VEL
LIN {X 0,Y 367.826,Z 898.203,A -85,B 0,C 180,E1 -12872.19,E2 -12872.19} C_VEL
LIN {X 0,Y 368.46,Z 892.738,A -85,B 0,C 180,E1 -12874.376,E2 -12874.376} C_VEL
LIN {X 0,Y 369.038,Z 887.571,A -85,B 0,C 180,E1 -12876.012,E2 -12876.012} C_VEL
LIN {X 0,Y 369.954,Z 880.119,A -85,B 0,C 180,E1 -12877.917,E2 -12877.917} C_VEL
LIN {X 0,Y 370.68,Z 871.98,A -85,B 0,C 180,E1 -12879.627,E2 -12879.627} C_VEL
LIN {X 0,Y 371.904,Z 863.037,A -85,B 0,C 180,E1 -12881.169,E2 -12881.169} C_VEL
LIN {X 0,Y 373.173,Z 852.694,A -85,B 0,C 180,E1 -12882.647,E2 -12882.647} C_VEL
LIN {X 0,Y 374.362,Z 841.628,A -85,B 0,C 180,E1 -12883.951,E2 -12883.951} C_VEL
LIN {X 0,Y 374.256,Z 836.869,A -85,B 0,C 180,E1 -12884.471,E2 -12884.471} C_VEL
LIN {X 0,Y 372.286,Z 828.978,A -85,B 0,C 180,E1 -12885.338,E2 -12885.338} C_VEL
LIN {X 0,Y 370.35,Z 820.73,A -85,B 0,C 180,E1 -12886.148,E2 -12886.148} C_VEL
LIN {X 0,Y 370.111,Z 815.428,A -85,B 0,C 180,E1 -12886.554,E2 -12886.554} C_VEL
LIN {X 0,Y 371.064,Z 801.487,A -85,B 0,C 180,E1 -12887.356,E2 -12887.356} C_VEL
LIN {X 0,Y 371.727,Z 787.401,A -85,B 0,C 180,E1 -12887.928,E2 -12887.928} C_VEL
LIN {X 0,Y 372.177,Z 772.573,A -85,B 0,C 180,E1 -12888.297,E2 -12888.297} C_VEL
LIN {X 0,Y 374.102,Z 674.794,A -85,B 0,C 180,E1 -12890.173,E2 -12890.173} C_VEL
LIN {X 0,Y 372.72,Z 669.434,A -85,B 0,C 180,E1 -12890.376,E2 -12890.376} C_VEL
LIN {X 0,Y 365.153,Z 650.283,A -85,B 0,C 180,E1 -12891.305,E2 -12891.305} C_VEL
LIN {X 0,Y 363.181,Z 645.404,A -85,B 0,C 180,E1 -12891.572,E2 -12891.572} C_VEL
LIN {X 0,Y 361.902,Z 639.532,A -85,B 0,C 180,E1 -12893.233,E2 -12893.233} C_VEL
LIN {X 0,Y 361.83,Z 639.539,A -85,B 0,C 180,E1 -12896.685,E2 -12896.685} C_VEL
LIN {X 0,Y 361.85,Z 639.538,A -85,B 0,C 180,E1 -12900.33,E2 -12900.33} C_VEL
LIN {X 0,Y 361.853,Z 639.536,A -85,B 0,C 180,E1 -12904.281,E2 -12904.281} C_VEL
LIN {X 0,Y 361.86,Z 639.536,A -85,B 0,C 180,E1 -12907.221,E2 -12907.221} C_VEL
LIN {X 0,Y 361.815,Z 639.529,A -85,B 0,C 180,E1 -12910.751,E2 -12910.751} C_VEL
LIN {X 0,Y 361.814,Z 639.535,A -85,B 0,C 180,E1 -12914.369,E2 -12914.369} C_VEL
LIN {X 0,Y 361.828,Z 639.538,A -85,B 0,C 180,E1 -12917.57,E2 -12917.57} C_VEL
LIN {X 0,Y 361.845,Z 639.519,A -85,B 0,C 180,E1 -12921.572,E2 -12921.572} C_VEL
LIN {X 0,Y 361.873,Z 639.521,A -85,B 0,C 180,E1 -12924.656,E2 -12924.656} C_VEL
LIN {X 0,Y 361.841,Z 639.533,A -85,B 0,C 180,E1 -12928.37,E2 -12928.37} C_VEL
LIN {X 0,Y 361.869,Z 639.526,A -85,B 0,C 180,E1 -12930.952,E2 -12930.952} C_VEL
LIN {X 0,Y 361.884,Z 639.527,A -85,B 0,C 180,E1 -12934.706,E2 -12934.706} C_VEL
LIN {X 0,Y 361.863,Z 639.531,A -85,B 0,C 180,E1 -12938.345,E2 -12938.345} C_VEL
LIN {X 0,Y 361.923,Z 639.51,A -85,B 0,C 180,E1 -12942.084,E2 -12942.084} C_VEL
LIN {X 0,Y 361.965,Z 639.521,A -85,B 0,C 180,E1 -12945.379,E2 -12945.379} C_VEL
LIN {X 0,Y 361.973,Z 639.51,A -85,B 0,C 180,E1 -12948.804,E2 -12948.804} C_VEL
LIN {X 0,Y 362.08,Z 639.506,A -85,B 0,C 180,E1 -12952.191,E2 -12952.191} C_VEL
LIN {X 0,Y 362.1,Z 639.501,A -85,B 0,C 180,E1 -12954.431,E2 -12954.431} C_VEL
LIN {X 0,Y 362.28,Z 639.484,A -85,B 0,C 180,E1 -12957.776,E2 -12957.776} C_VEL
LIN {X 0,Y 362.427,Z 639.459,A -85,B 0,C 180,E1 -12960,E2 -12960} C_VEL
LIN {X 0,Y 362.282,Z 639.482,A -85,B 0,C 180,E1 -12962.223,E2 -12962.223} C_VEL
LIN {X 0,Y 362.149,Z 639.494,A -85,B 0,C 180,E1 -12966.686,E2 -12966.686} C_VEL
LIN {X 0,Y 362.058,Z 639.507,A -85,B 0,C 180,E1 -12968.933,E2 -12968.933} C_VEL
LIN {X 0,Y 361.963,Z 639.522,A -85,B 0,C 180,E1 -12972.332,E2 -12972.332} C_VEL
LIN {X 0,Y 361.965,Z 639.515,A -85,B 0,C 180,E1 -12974.62,E2 -12974.62} C_VEL
LIN {X 0,Y 361.962,Z 639.522,A -85,B 0,C 180,E1 -12978.099,E2 -12978.099} C_VEL
LIN {X 0,Y 361.863,Z 639.531,A -85,B 0,C 180,E1 -12981.655,E2 -12981.655} C_VEL
LIN {X 0,Y 361.928,Z 639.522,A -85,B 0,C 180,E1 -12985.29,E2 -12985.29} C_VEL
LIN {X 0,Y 361.92,Z 639.521,A -85,B 0,C 180,E1 -12987.778,E2 -12987.778} C_VEL
LIN {X 0,Y 361.849,Z 639.532,A -85,B 0,C 180,E1 -12991.285,E2 -12991.285} C_VEL
LIN {X 0,Y 361.857,Z 639.534,A -85,B 0,C 180,E1 -12994.28,E2 -12994.28} C_VEL
LIN {X 0,Y 361.867,Z 639.531,A -85,B 0,C 180,E1 -12997.223,E2 -12997.223} C_VEL
LIN {X 0,Y 361.874,Z 639.534,A -85,B 0,C 180,E1 -13000.762,E2 -13000.762} C_VEL
LIN {X 0,Y 361.866,Z 639.533,A -85,B 0,C 180,E1 -13004.361,E2 -13004.361} C_VEL
LIN {X 0,Y 361.838,Z 639.534,A -85,B 0,C 180,E1 -13007.568,E2 -13007.568} C_VEL
LIN {X 0,Y 361.873,Z 639.536,A -85,B 0,C 180,E1 -13010.973,E2 -13010.973} C_VEL
LIN {X 0,Y 361.876,Z 639.536,A -85,B 0,C 180,E1 -13014.655,E2 -13014.655} C_VEL
LIN {X 0,Y 361.883,Z 639.621,A -85,B 0,C 180,E1 -13016.789,E2 -13016.789} C_VEL
LIN {X 0,Y 365.321,Z 654.118,A -85,B 0,C 180,E1 -13020.253,E2 -13020.253} C_VEL
LIN {X 0,Y 367.468,Z 664.776,A -85,B 0,C 180,E1 -13022.676,E2 -13022.676} C_VEL
LIN {X 0,Y 367.105,Z 669.948,A -85,B 0,C 180,E1 -13023.738,E2 -13023.738} C_VEL
LIN {X 0,Y 373.652,Z 708.615,A -85,B 0,C 180,E1 -13024.986,E2 -13024.986} C_VEL
LIN {X 0,Y 371.749,Z 805.899,A -85,B 0,C 180,E1 -13026.866,E2 -13026.866} C_VEL
LIN {X 0,Y 371.084,Z 819.978,A -85,B 0,C 180,E1 -13027.301,E2 -13027.301} C_VEL
LIN {X 0,Y 370.051,Z 834.362,A -85,B 0,C 180,E1 -13027.97,E2 -13027.97} C_VEL
LIN {X 0,Y 368.872,Z 848.209,A -85,B 0,C 180,E1 -13028.867,E2 -13028.867} C_VEL
LIN {X 0,Y 367.676,Z 860.333,A -85,B 0,C 180,E1 -13029.875,E2 -13029.875} C_VEL
LIN {X 0,Y 366.293,Z 872.294,A -85,B 0,C 180,E1 -13031.108,E2 -13031.108} C_VEL
LIN {X 0,Y 365.075,Z 882.234,A -85,B 0,C 180,E1 -13032.35,E2 -13032.35} C_VEL
LIN {X 0,Y 363.719,Z 893.197,A -85,B 0,C 180,E1 -13034.017,E2 -13034.017} C_VEL
LIN {X 0,Y 362.642,Z 902.259,A -85,B 0,C 180,E1 -13035.696,E2 -13035.696} C_VEL
LIN {X 0,Y 361.897,Z 909.788,A -85,B 0,C 180,E1 -13037.38,E2 -13037.38} C_VEL
LIN {X 0,Y 361.116,Z 916.98,A -85,B 0,C 180,E1 -13039.345,E2 -13039.345} C_VEL
LIN {X 0,Y 360.748,Z 921.999,A -85,B 0,C 180,E1 -13041.034,E2 -13041.034} C_VEL
LIN {X 0,Y 360.484,Z 927.169,A -85,B 0,C 180,E1 -13043.282,E2 -13043.282} C_VEL
LIN {X 0,Y 360.361,Z 930.811,A -85,B 0,C 180,E1 -13045.526,E2 -13045.526} C_VEL
LIN {X 0,Y 360.313,Z 933.033,A -85,B 0,C 180,E1 -13047.764,E2 -13047.764} C_VEL
LIN {X 0,Y 360.422,Z 933.899,A -85,B 0,C 180,E1 -13050,E2 -13050} C_VEL
LIN {X 0,Y 360.294,Z 933.414,A -85,B 0,C 180,E1 -13052.236,E2 -13052.236} C_VEL
LIN {X 0,Y 360.359,Z 931.594,A -85,B 0,C 180,E1 -13054.474,E2 -13054.474} C_VEL
LIN {X 0,Y 360.485,Z 928.395,A -85,B 0,C 180,E1 -13056.717,E2 -13056.717} C_VEL
LIN {X 0,Y 360.769,Z 923.699,A -85,B 0,C 180,E1 -13058.966,E2 -13058.966} C_VEL
LIN {X 0,Y 361.345,Z 917.373,A -85,B 0,C 180,E1 -13061.215,E2 -13061.215} C_VEL
LIN {X 0,Y 362.274,Z 910.354,A -85,B 0,C 180,E1 -13063.176,E2 -13063.176} C_VEL
LIN {X 0,Y 363.409,Z 901.677,A -85,B 0,C 180,E1 -13065.134,E2 -13065.134} C_VEL
LIN {X 0,Y 364.668,Z 892.628,A -85,B 0,C 180,E1 -13066.803,E2 -13066.803} C_VEL
LIN {X 0,Y 366.22,Z 881.695,A -85,B 0,C 180,E1 -13068.46,E2 -13068.46} C_VEL
LIN {X 0,Y 367.82,Z 870.612,A -85,B 0,C 180,E1 -13069.825,E2 -13069.825} C_VEL
LIN {X 0,Y 369.392,Z 858.134,A -85,B 0,C 180,E1 -13071.073,E2 -13071.073} C_VEL
LIN {X 0,Y 370.867,Z 844.776,A -85,B 0,C 180,E1 -13072.125,E2 -13072.125} C_VEL
LIN {X 0,Y 372.167,Z 831.516,A -85,B 0,C 180,E1 -13072.922,E2 -13072.922} C_VEL
LIN {X 0,Y 373.216,Z 818.024,A -85,B 0,C 180,E1 -13073.514,E2 -13073.514} C_VEL
LIN {X 0,Y 373.871,Z 803.065,A -85,B 0,C 180,E1 -13073.949,E2 -13073.949} C_VEL
LIN {X 0,Y 375.98,Z 709.225,A -85,B 0,C 180,E1 -13075.764,E2 -13075.764} C_VEL
LIN {X 0,Y 371.612,Z 684.857,A -85,B 0,C 180,E1 -13076.636,E2 -13076.636} C_VEL
LIN {X 0,Y 368.444,Z 669.651,A -85,B 0,C 180,E1 -13077.245,E2 -13077.245} C_VEL
LIN {X 0,Y 368.347,Z 666.818,A -85,B 0,C 180,E1 -13077.869,E2 -13077.869} C_VEL
LIN {X 0,Y 365.843,Z 655.182,A -85,B 0,C 180,E1 -13080.663,E2 -13080.663} C_VEL
LIN {X 0,Y 362.76,Z 642.938,A -85,B 0,C 180,E1 -13083.784,E2 -13083.784} C_VEL
LIN {X 0,Y 361.892,Z 639.522,A -85,B 0,C 180,E1 -13084.698,E2 -13084.698} C_VEL
LIN {X 0,Y 361.874,Z 639.531,A -85,B 0,C 180,E1 -13088.424,E2 -13088.424} C_VEL
LIN {X 0,Y 361.855,Z 639.531,A -85,B 0,C 180,E1 -13091.327,E2 -13091.327} C_VEL
LIN {X 0,Y 361.823,Z 639.531,A -85,B 0,C 180,E1 -13094.368,E2 -13094.368} C_VEL
LIN {X 0,Y 361.856,Z 639.523,A -85,B 0,C 180,E1 -13097.565,E2 -13097.565} C_VEL
LIN {X 0,Y 361.876,Z 639.532,A -85,B 0,C 180,E1 -13100.972,E2 -13100.972} C_VEL
LIN {X 0,Y 361.875,Z 639.53,A -85,B 0,C 180,E1 -13104.655,E2 -13104.655} C_VEL
LIN {X 0,Y 361.837,Z 639.512,A -85,B 0,C 180,E1 -13108.371,E2 -13108.371} C_VEL
LIN {X 0,Y 361.9,Z 639.524,A -85,B 0,C 180,E1 -13110.955,E2 -13110.955} C_VEL
LIN {X 0,Y 361.955,Z 639.518,A -85,B 0,C 180,E1 -13113.475,E2 -13113.475} C_VEL
LIN {X 0,Y 361.891,Z 639.525,A -85,B 0,C 180,E1 -13117.145,E2 -13117.145} C_VEL
LIN {X 0,Y 361.922,Z 639.522,A -85,B 0,C 180,E1 -13120.724,E2 -13120.724} C_VEL
LIN {X 0,Y 361.95,Z 639.525,A -85,B 0,C 180,E1 -13124.227,E2 -13124.227} C_VEL
LIN {X 0,Y 362,Z 639.511,A -85,B 0,C 180,E1 -13126.528,E2 -13126.528} C_VEL
